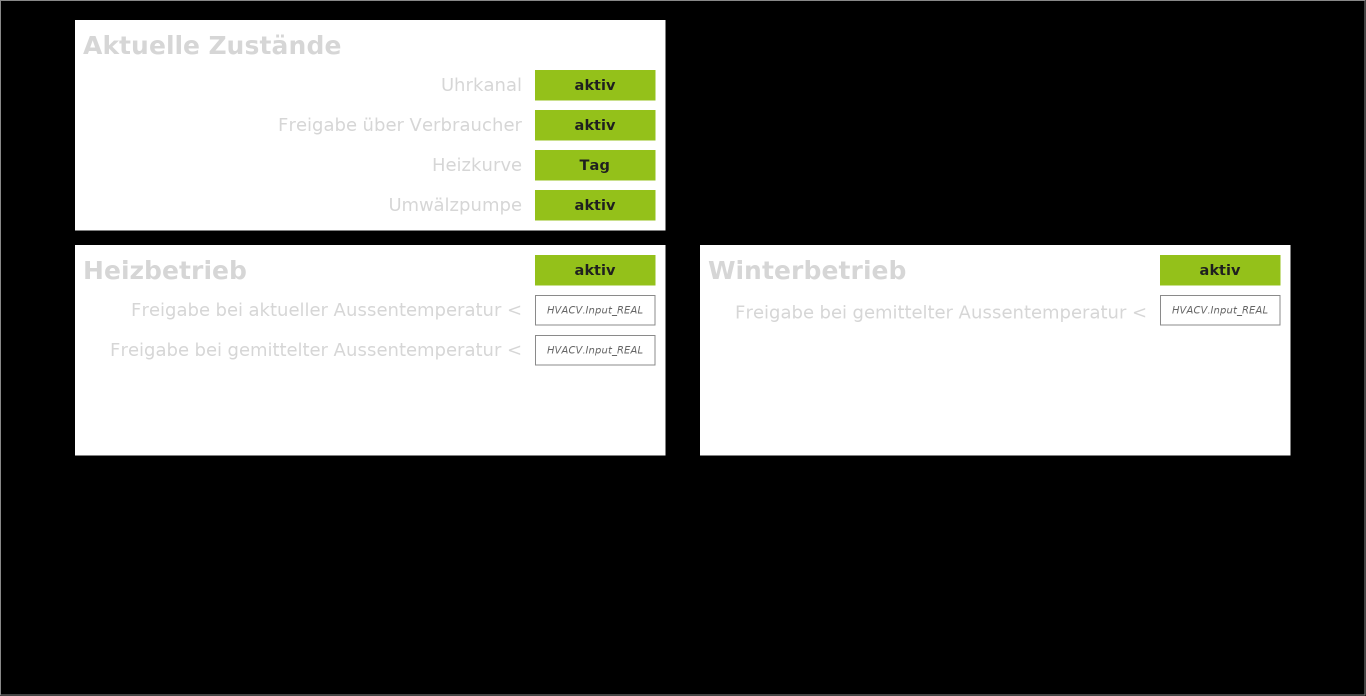
VISUALIZATION HeatingCircuit_VenA_Settings  // 1366x696
VAR_IN_OUT
	FB : HeatingCircuit_VenA;
END_VAR
    Rectangle (75,245 590x210)
    Rectangle (80,250 435x40), "Heizbetrieb"
    Rectangle (75,295 450x30), "Freigabe bei aktueller Aussentemperatur <"
    Rectangle (75,335 450x30), "Freigabe bei gemittelter Aussentemperatur <"
    RoundedRectangle (535,255 120x30), "inaktiv", invisible if: FB.HEAT
    RoundedRectangle (535,255 120x30), "aktiv", invisible if: NOT FB.HEAT
    Rectangle (75,20 590x210)
    Rectangle (80,25 570x40), "Aktuelle Zustände"
    Rectangle (75,70 450x30), "Uhrkanal"
    Rectangle (75,110 450x30), "Freigabe über Verbraucher"
    RoundedRectangle (535,70 120x30), "inaktiv", invisible if: FB.Clock_Channel
    RoundedRectangle (535,70 120x30), "aktiv", invisible if: NOT FB.Clock_Channel
    RoundedRectangle (535,110 120x30), "inaktiv", invisible if: FB.EXT_REQ
    RoundedRectangle (535,110 120x30), "aktiv", invisible if: NOT FB.EXT_REQ
    Rectangle (75,150 450x30), "Heizkurve"
    Rectangle (75,190 450x30), "Umwälzpumpe"
    RoundedRectangle (535,150 120x30), "Nacht", invisible if: FB.MODE
    RoundedRectangle (535,150 120x30), "Tag", invisible if: NOT FB.MODE
    RoundedRectangle (535,190 120x30), "inaktiv", invisible if: FB.pump.xAB
    RoundedRectangle (535,190 120x30), "aktiv", invisible if: NOT FB.pump.xAB
    Line (75,225)
    Line (965,345)
    Rectangle (700,245 590x210)
    Rectangle (705,250 435x40), "Winterbetrieb"
    Rectangle (700,295 450x35), "Freigabe bei gemittelter Aussentemperatur <"
    RoundedRectangle (1160,255 120x30), "inaktiv", invisible if: FB.WINTER
    RoundedRectangle (1160,255 120x30), "aktiv", invisible if: NOT FB.WINTER
    Frame (535,295 120x30)
        shows HVACV.Input_REAL(rValue := FB.Setpoint_Heat_Act.rSetPoint, bDecimals := 1, sUnit := '°C', rMinInputVisu := -20, rMaxInputVisu := 50, sDialogTitle := 'Release actual outsidetemp.')
    Frame (535,335 120x30)
        shows HVACV.Input_REAL(rValue := FB.Setpoint_Heat_Aver.rSetPoint, bDecimals := 1, sUnit := '°C', rMinInputVisu := -20, rMaxInputVisu := 50, sDialogTitle := 'Release average outsidetemp.')
    Frame (1160,295 120x30)
        shows HVACV.Input_REAL(rValue := FB.Setpoint_WINTER.rSetPoint, bDecimals := 1, sUnit := '°C', rMinInputVisu := -20, rMaxInputVisu := 50, sDialogTitle := 'Release winter operation')
END_VISUALIZATION

// Device/Application/Macros and frames/HeatingCircuit/Pump_Frames/Pump_Button
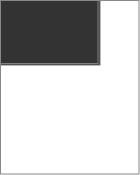
VISUALIZATION Pump_Button  // 140x175
VAR_IN_OUT
	FB_Pump : HVAC.Pump;
END_VAR

VAR 
	
END_VAR
    Rectangle (0,0 100x65), invisible if: TRUE
    Button (0,0 100x65)
        OnMouseClick:  Dialog=Pump_Parameter_Dialog, Parameters={FB_Pump: FB_Pump}, Selected={1: }, OpenModal=True, OpenCentered=True
END_VISUALIZATION

// Device/Application/Visu/1_Objects/HC_1/Heatcurve_HC_1
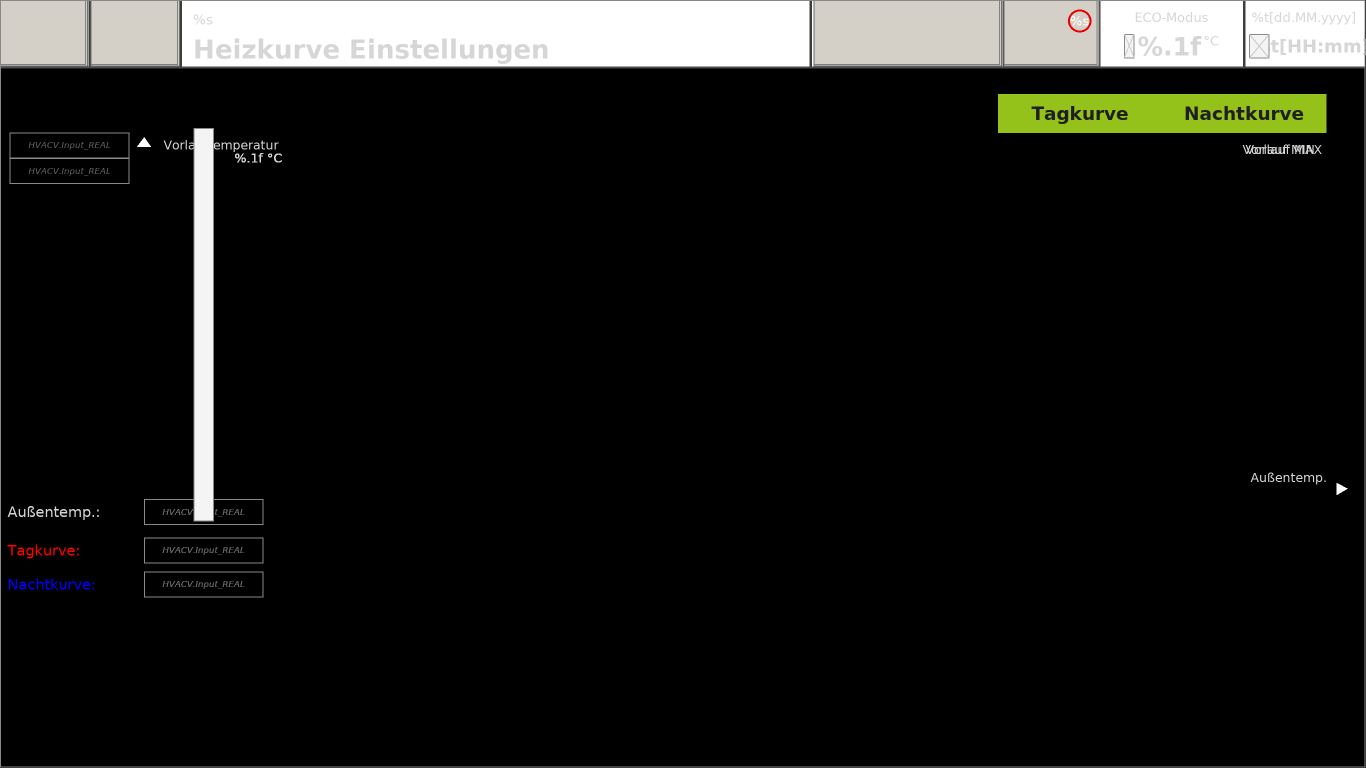
VISUALIZATION Heatcurve_HC_1  // 1366x768
    Frame (0,0 1366x70)
        shows Header_Frame()
    Rectangle (190,5 545x30), "%s", text variable: CONCAT( CONCAT(PRG.GebVar, ' | Start | Objekte | '), Prg.HC_1.Title)
    Rectangle (190,32 545x35), "Heizkurve Einstellungen"
    Frame (0,90 1357x595)
        shows HeatCurve4P_DN(FB_HeatCurve4P_DN := PRG.HC_1.HC)
END_VISUALIZATION

// Device/Application/Visu/1_Objects/HC_1/Trend_HC_1
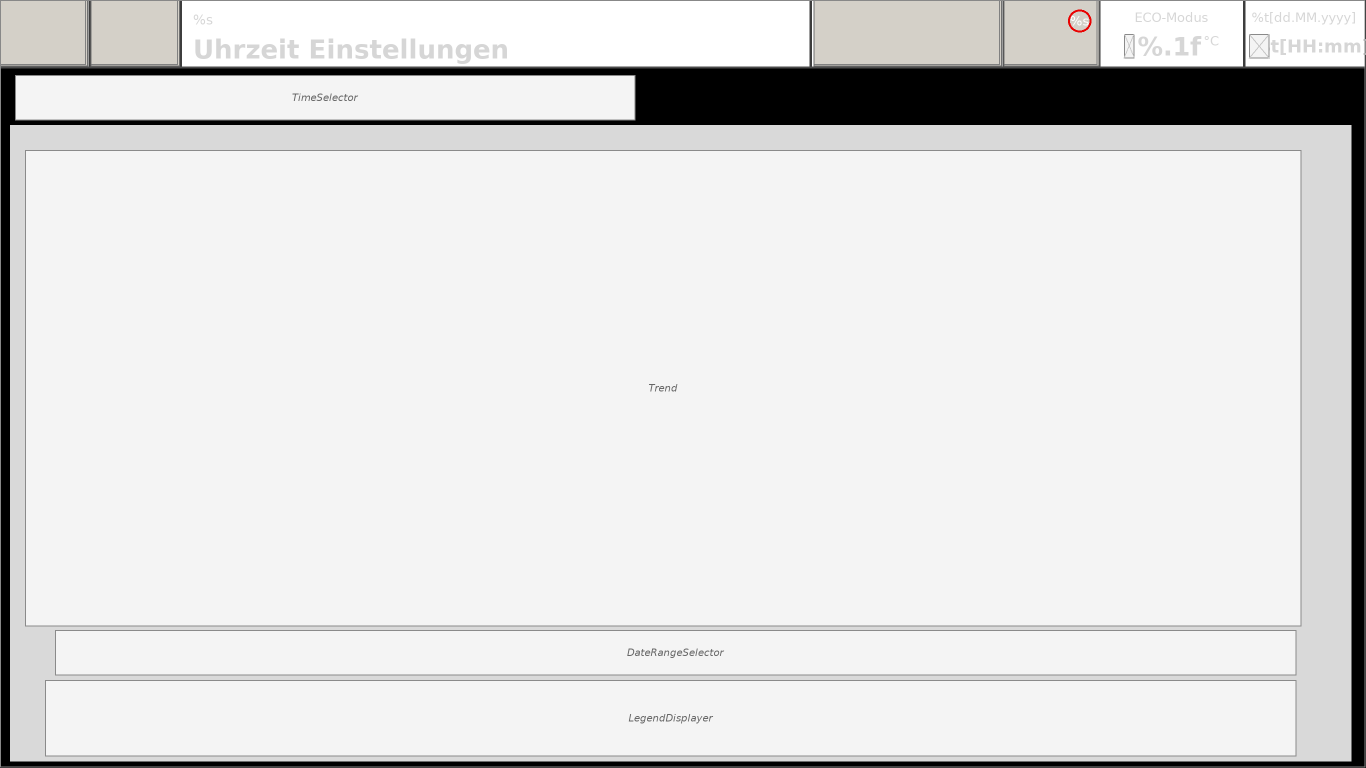
VISUALIZATION Trend_HC_1  // 1366x768
    Rectangle (10,125 1341x636)
    Frame (0,0 1366x70)
        shows Header_Frame()
    Rectangle (190,5 545x30), "%s", text variable: CONCAT( CONCAT(PRG.GebVar, ' | Start | Objekte | '), Prg.HC_1.Title)
    Rectangle (190,32 545x35), "Uhrzeit Einstellungen", text variable: PRG.HC_1.Title
    Trend (25,150 1276x476)
        p758368661: dd.MM.yyyy
        p2423372160: HH:mm
        p2833066001: HC_1_Trend
        p2059293862: Trend1DateRangeSelector
        p2541140726: Trend1TimeSelector
        p1690078355: Trend1Legend
    DateRangeSelector (55,630 1241x45)
        p758368661: dd.MM
        p2423372160: HH:mm
        p1661464551: GenElemInst_54
    TimeSelector (15,75 620x45)
        p3737533738: GenElemInst_54
        p677259794: Zoom:
    LegendDisplayer (45,680 1251x76)
        p3773266362: GenElemInst_54
END_VISUALIZATION

// Device/Application/Visu/3_Settings/Settings_MANInfo
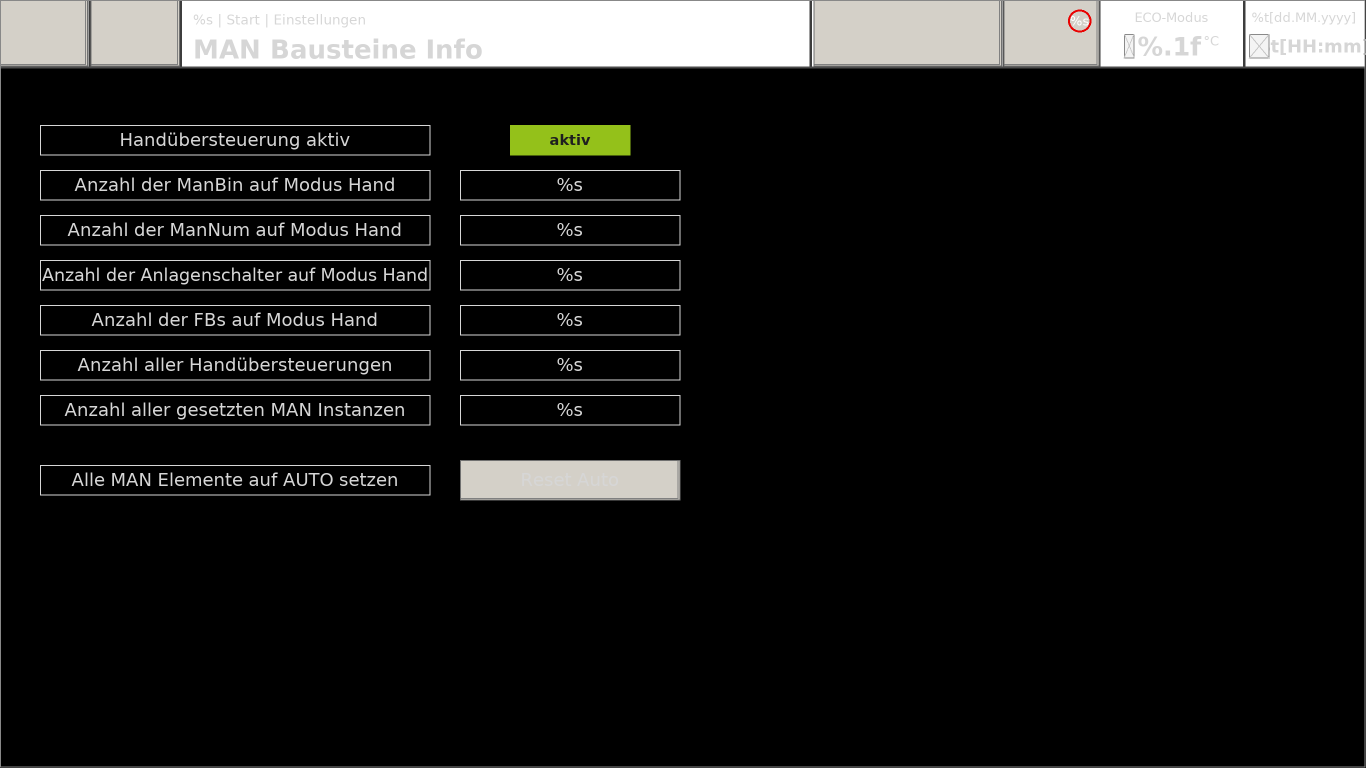
VISUALIZATION Settings_MANInfo  // 1366x768
    Rectangle (460,170 220x30), "%s", text variable: Main.ManInfo.iManBinCounter
    Rectangle (460,215 220x30), "%s", text variable: Main.ManInfo.iManNumCounter
    Rectangle (460,260 220x30), "%s", text variable: Main.ManInfo.iManOpCounter
    Rectangle (460,305 220x30), "%s", text variable: Main.ManInfo.iManFbCounter
    Rectangle (460,395 220x30), "%s", text variable: Main.ManInfo.iManCounter
    Rectangle (40,125 390x30), "Handübersteuerung aktiv"
    Rectangle (40,170 390x30), "Anzahl der ManBin auf Modus Hand"
    Rectangle (40,215 390x30), "Anzahl der ManNum auf Modus Hand"
    Rectangle (40,260 390x30), "Anzahl der Anlagenschalter auf Modus Hand"
    Rectangle (40,305 390x30), "Anzahl der FBs auf Modus Hand"
    Rectangle (40,395 390x30), "Anzahl aller gesetzten MAN Instanzen"
    Button (460,460 220x40), "Reset Auto"
        toggle Main.ManInfo.xResetAuto
    Frame (0,0 1366x70)
        shows Header_Frame()
    Rectangle (190,5 545x30), "%s | Start | Einstellungen", text variable: PRG.GebVar
    Rectangle (190,32 545x35), "MAN Bausteine Info"
    RoundedRectangle (510,125 120x30), "inaktiv", invisible if: Main.ManInfo.xManActive
    RoundedRectangle (510,125 120x30), "aktiv", invisible if: NOT Main.ManInfo.xManActive
    Rectangle (460,350 220x30), "%s", text variable: Main.ManInfo.iManCounter
    Rectangle (40,350 390x30), "Anzahl aller Handübersteuerungen"
    Rectangle (40,465 390x30), "Alle MAN Elemente auf AUTO setzen"
END_VISUALIZATION

// Device/Application/Visu/1_Objects/HC_1/Clock_HC_1
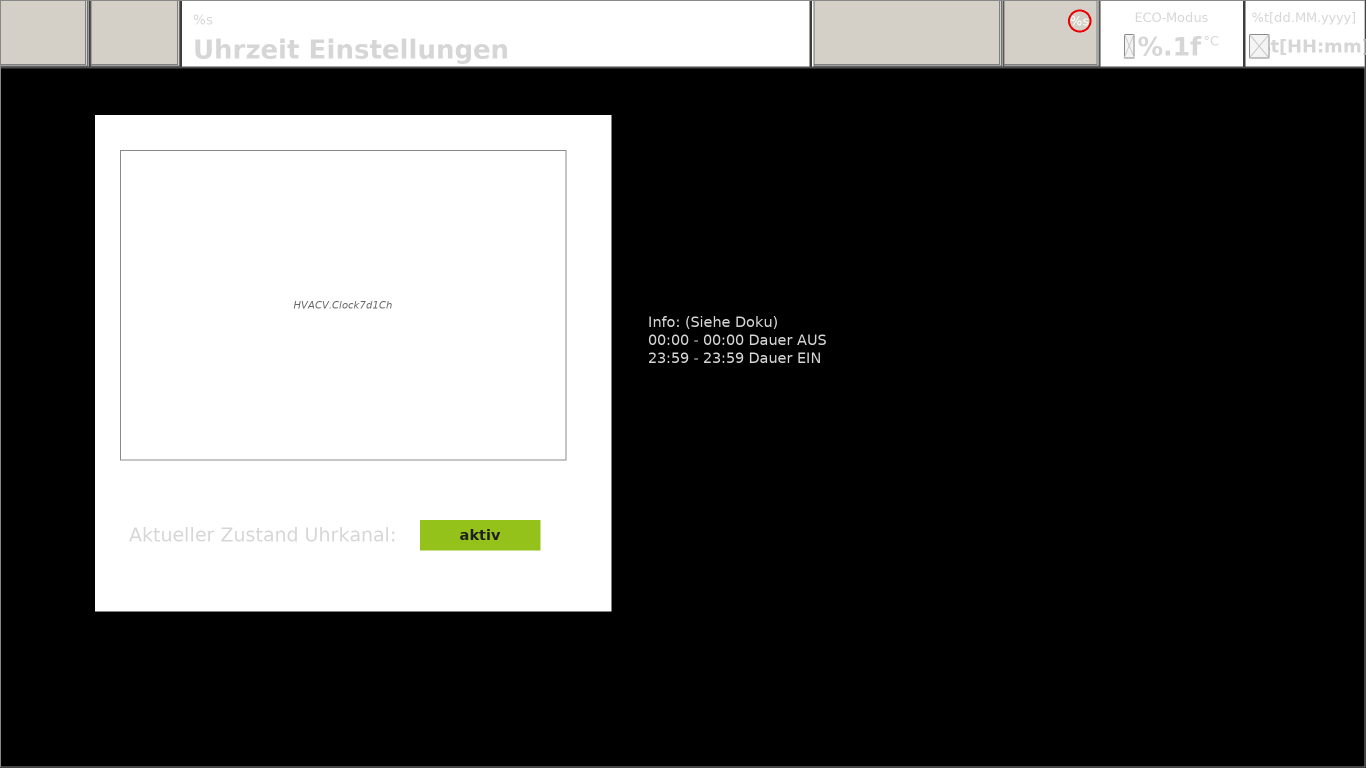
VISUALIZATION Clock_HC_1  // 1366x768
    Rectangle (95,115 516x496)
    Frame (0,0 1366x70)
        shows Header_Frame()
    Rectangle (190,5 545x30), "%s", text variable: CONCAT( CONCAT(PRG.GebVar, ' | Start | Objekte | '), Prg.HC_1.Title)
    Rectangle (190,32 545x35), "Uhrzeit Einstellungen", text variable: PRG.HC_1.Title
    RoundedRectangle (420,520 120x30), "inaktiv", invisible if: PRG.HC_1.Clock.xActive
    RoundedRectangle (420,520 120x30), "aktiv", invisible if: NOT PRG.HC_1.Clock.xActive
    Rectangle (115,520 296x30), "Aktueller Zustand Uhrkanal:"
    Frame (120,150 446x310)
        shows HVACV.Clock7d1Ch(FB_Clock7d1Ch := PRG.HC_1.Clock)
    Rectangle (645,295 447x90), "Info: (Siehe Doku) 00:00 - 00:00 Dauer AUS 23:59 - 23:59 Dauer EIN"
END_VISUALIZATION

// Device/Application/Visu/1_Objects/Room_1/Start_Room_1
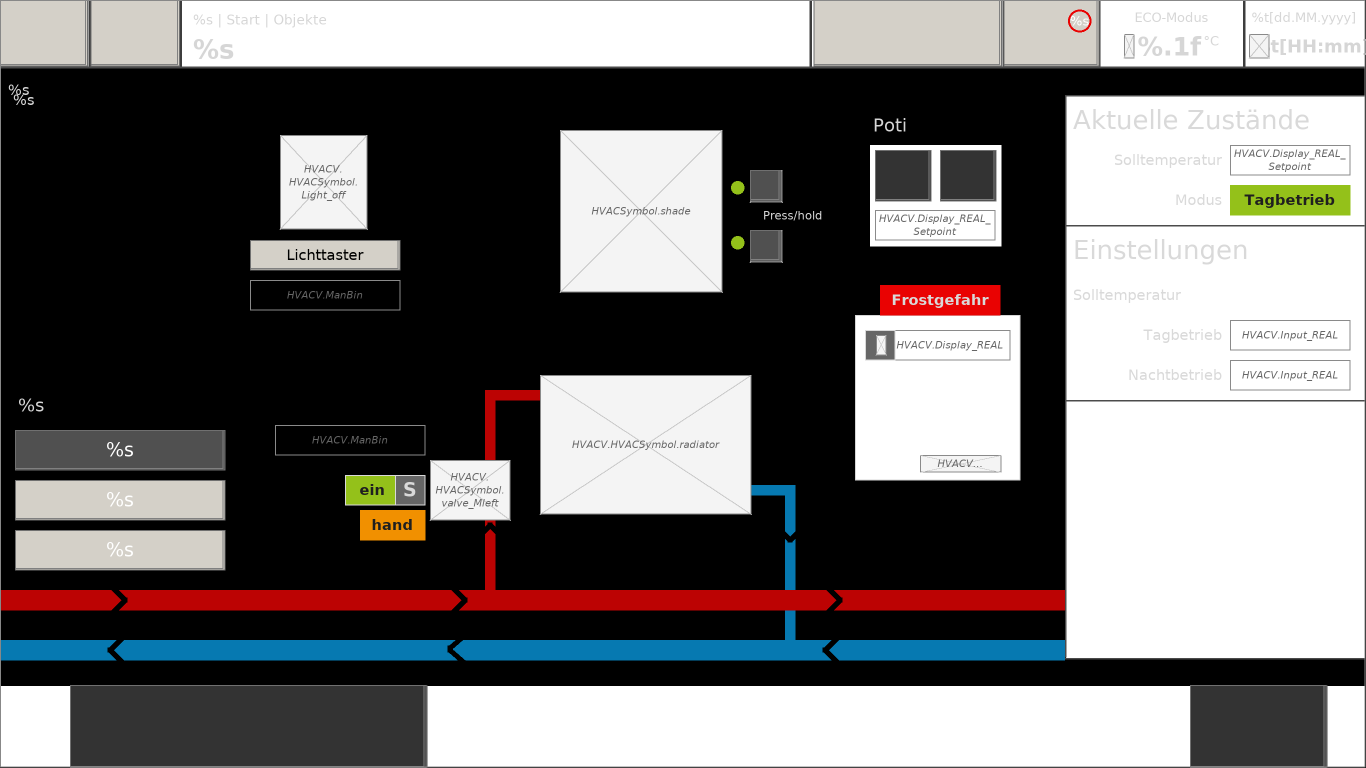
VISUALIZATION Start_Room_1  // 1366x768
    Frame (0,70 1366x613)
        shows Zone_F_Therm_Start(FB := PRG.Room_1)
    Frame (0,0 1366x70)
        shows Header_Frame()
    Rectangle (190,5 545x30), "%s | Start | Objekte", text variable: PRG.GebVar
    Rectangle (190,32 545x35), "%s", text variable: PRG.Room_1.Titel
    Rectangle (0,685 1366x83)
    Rectangle (425,685 2x83)
    Rectangle (70,685 2x83)
    Rectangle (130,685 166x83), "ZEITSCHALTUNG"
    Image (80,710 36x35), image: HVACV.HVACImage.clock
    RoundedRectangle (295,715 120x30), "inaktiv", invisible if: PRG.Room_1.Clock.xActive
    RoundedRectangle (295,715 120x30), "aktiv", invisible if: NOT PRG.Room_1.Clock.xActive
    Button (70,685 356x83)
        OnMouseClick:  Assign=Clock_Room_1, Type=Assignment
    Rectangle (1190,685 2x83)
    Rectangle (1325,685 2x83)
    Rectangle (1260,685 71x83), "HILFE"
    Image (1205,705 31x47), image: HVACV.HVACImage.help
    Button (1190,685 136x83)
        OnMouseClick:  Dialog=HVACV.Help_Start, OpenModal=True, OpenCentered=True
    Rectangle (10,85 536x30), "%s", text variable: PRG.Room_Line1.sSetPoint
        OnMouseClick: write the text variable via Default
END_VISUALIZATION

// Device/Application/Macros and frames/HeatingCircuit/Valve_Frames/ValveAnalog_Button
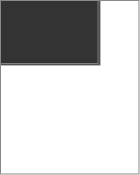
VISUALIZATION ValveAnalog_Button  // 140x175
VAR_IN_OUT
	FB_ValveAnalog : HVAC.ValveAnalog;
END_VAR

VAR 
	
END_VAR
    Rectangle (0,0 100x65), invisible if: TRUE
    Button (0,0 100x65)
        OnMouseClick:  Dialog=ValveAnalog_Parameter_Dialog, Parameters={FB_ValveAnalog: FB_ValveAnalog}, Selected={1: }, OpenModal=True, OpenCentered=True
END_VISUALIZATION

// Device/Application/Macros and frames/HeatingCircuit/HeatingCircuit_VenA
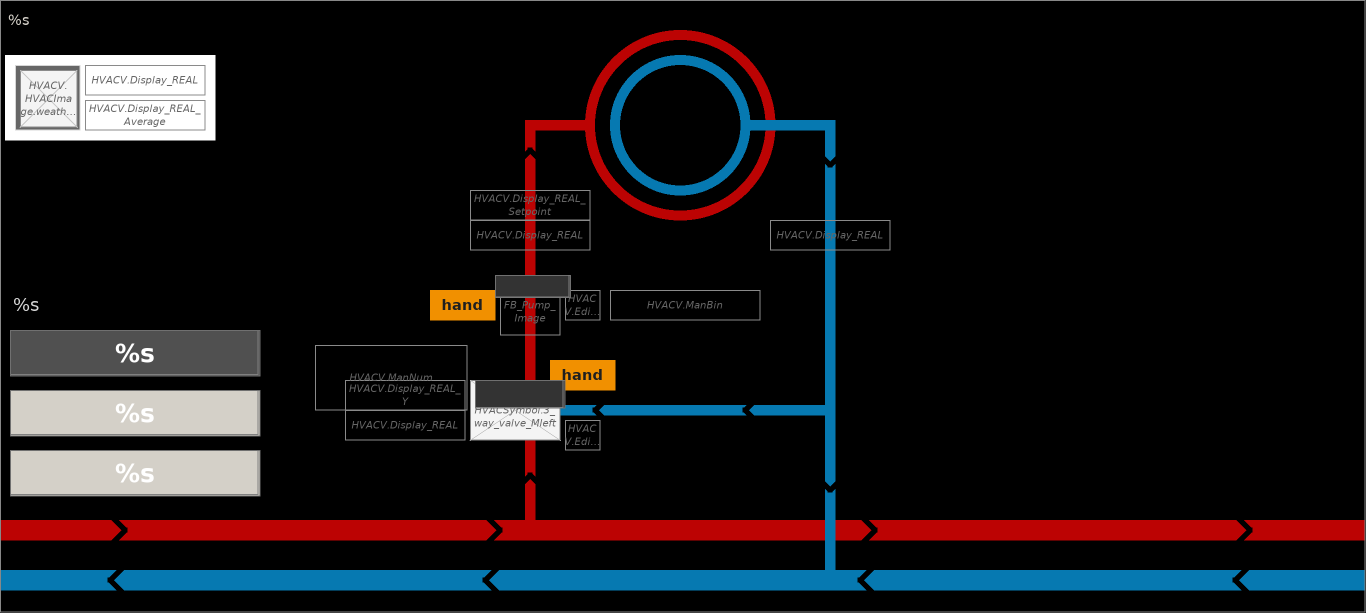
VISUALIZATION HeatingCircuit_VenA  // 1366x613
VAR_IN_OUT
	FB : HeatingCircuit_VenA;
END_VAR
    Rectangle (5,0 970x40), "%s", text variable: FB.Line1
    Rectangle (0,520 1365x20)
    Rectangle (0,570 1365x20)
    Polyline (875,565) (860,580) (875,595)
    Polyline (860,515) (875,530) (860,545)
    Polyline (125,565) (110,580) (125,595)
    Polyline (110,515) (125,530) (110,545)
    Polyline (485,515) (500,530) (485,545)
    Line (335,515)
    Polyline (1250,565) (1235,580) (1250,595)
    Polyline (1235,515) (1250,530) (1235,545)
    Rectangle (525,430 10x100)
    Rectangle (825,120 10x460)
    Rectangle (545,405 285x10)
    Rectangle (525,120 10x270)
    Polyline (515,490) (530,475) (545,490)
    Polyline (815,475) (830,490) (845,475)
    Polyline (815,150) (830,165) (845,150)
    Polyline (610,395) (595,410) (610,425)
    Polyline (760,395) (745,410) (760,425)
    Rectangle (525,120 65x10)
    Polyline (515,165) (530,150) (545,165)
    Image (470,380 90x60), image: HVACV.HVACSymbol.3_way_valve_Mleft
    Group (585,30 190x190)
        Ellipse (0,0 190x190)
        Ellipse (10,10 170x170)
        Ellipse (25,25 140x140)
        Ellipse (35,35 120x120)
    Rectangle (745,120 90x10)
    RoundedRectangle (430,290 65x30), "hand", invisible if: FB.Pump_AOO=0
    RoundedRectangle (550,360 65x30), "hand", invisible if: FB.Valve_AO = 0
    Frame (565,420 35x30)
        shows HVACV.Edit_symbol()
    Polyline (500,565) (485,580) (500,595)
    Frame (470,190 120x30)
        shows HVACV.Display_REAL_Setpoint(rSetpoint := FB.Setpoint_FT, bDecimals := 1, xAlarm := FALSE, sUnit := '°C')
    Frame (565,290 35x30)
        shows HVACV.Edit_symbol()
    Frame (500,275 60x60)
        shows HVACV.FB_Pump_Image(FB_Pump := FB.Pump)
    Rectangle (5,55 210x85)
    RoundedRectangle (15,65 65x65)
    Image (20,70 57x57), image: HVACV.HVACImage.weather
    Frame (85,100 120x30)
        shows HVACV.Display_REAL_Average(rValue := FB.OutTempAverage, bDecimals := 1, xAlarm := FALSE, sUnit := '°C')
    Frame (470,220 120x30)
        shows HVACV.Display_REAL(rValue := FB.TS_FT, bDecimals := 1, xAlarm := FB.TS_FT_ERR, sUnit := '°C')
    Frame (610,290 150x30)
        shows HVACV.ManBin(eManModeB := FB.Pump.eManModeB)
    Frame (85,65 120x30)
        shows HVACV.Display_REAL(rValue := FB.OutTemp, bDecimals := 1, xAlarm := FALSE, sUnit := '°C')
    Frame (770,220 120x30)
        shows HVACV.Display_REAL(rValue := FB.TS_RT, bDecimals := 1, xAlarm := FB.TS_RT_ERR, sUnit := '°C')
    Button (10,330 250x46), "%s", text variable: FB.OS.sTitleM0, colour toggle: FB.OS.eMode = 0
        OnMouseClick: execute { FB.OS.eMode := 0; }
    Button (10,390 250x46), "%s", text variable: FB.OS.sTitleM1, colour toggle: FB.OS.eMode =1
        OnMouseClick: execute { FB.OS.eMode := 1; }
    Button (10,450 250x46), "%s", text variable: FB.OS.sTitleM2, colour toggle: FB.OS.eMode =2
        OnMouseClick: execute { FB.OS.eMode := 2; }
    Frame (495,275 106x61)
        shows Pump_Button(FB_Pump := FB.Pump)
    Rectangle (10,290 250x30), "%s", text variable: FB.OS.sTitle
    Frame (475,380 126x76)
        shows ValveAnalog_Button(FB_ValveAnalog := FB.Valve)
    Frame (345,380 120x30)
        shows HVACV.Display_REAL_Y(rValue := FB.Valve_HA, bDecimals := 1, sUnit := '%')
    Frame (345,410 120x30)
        shows HVACV.Display_REAL(rValue := FB.Valve_rU, bDecimals := 1, xAlarm := FB.Valve.xAlarm, sUnit := '%')
    Frame (315,345 152x65)
        shows HVACV.ManNum(eManModeN := FB.Valve.eManModeN, rManValue := FB.Valve.rManValue, bDecimals := 1, sUnit := '%', rMinInputVisu := 0, rMaxInputVisu := 100, sDialogTitle := 'Manual valve position')
END_VISUALIZATION

// Device/Application/Visu/1_Objects/HC_1/Start_HC_1
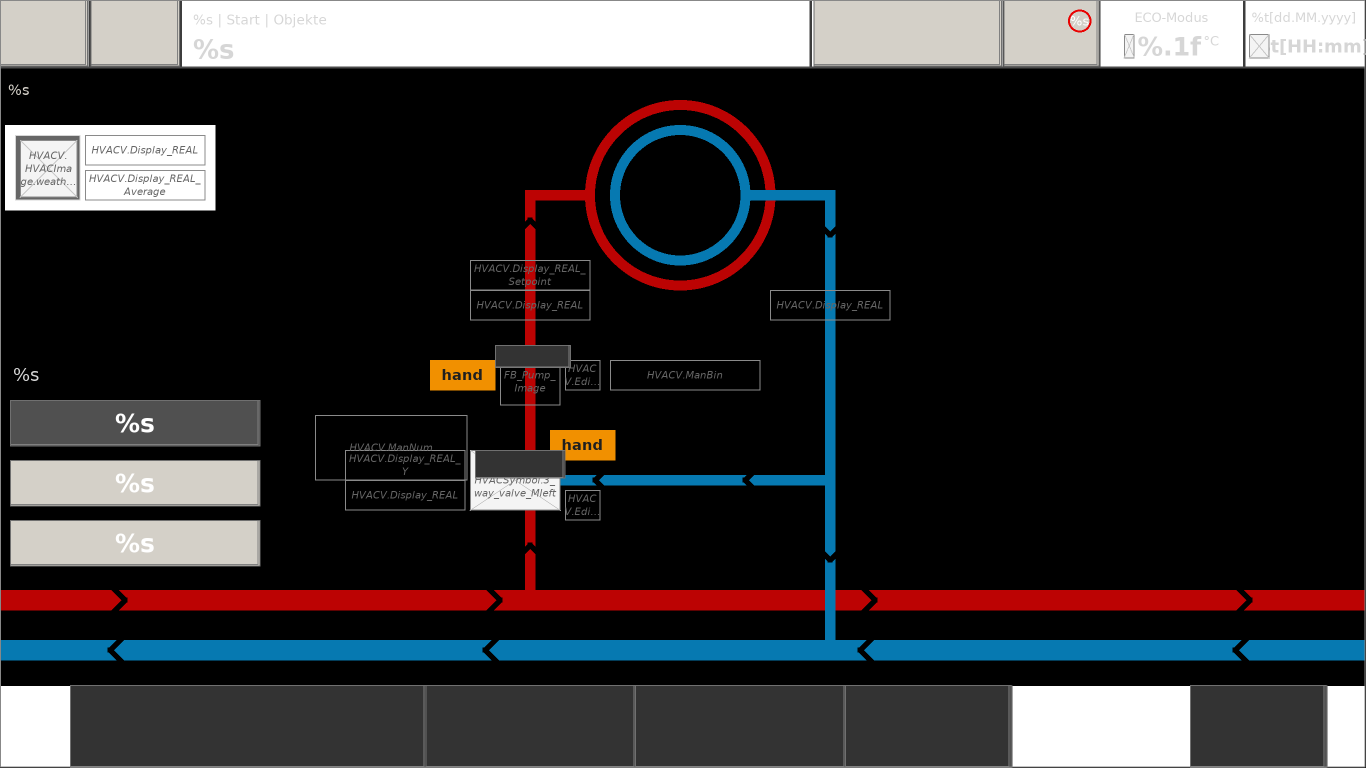
VISUALIZATION Start_HC_1  // 1366x768
    Frame (0,0 1366x70)
        shows Header_Frame()
    Rectangle (190,5 545x30), "%s | Start | Objekte", text variable: PRG.GebVar
    Rectangle (190,32 545x35), "%s", text variable: PRG.HC_1.Title
    Rectangle (0,685 1366x83)
    Rectangle (635,685 2x83)
    Rectangle (425,685 2x83)
    Rectangle (500,685 135x83), "EINSTELLUNG"
    Image (440,705 46x36), image: HVACV.HVACImage.settings
    Button (425,685 211x83)
        OnMouseClick:  Assign=Settings_HC_1, Type=Assignment
    Frame (0,70 1366x613)
        shows HeatingCircuit_VenA(FB := PRG.HC_1)
    Rectangle (70,685 2x83)
    Rectangle (130,685 166x83), "ZEITSCHALTUNG"
    Image (80,710 36x35), image: HVACV.HVACImage.clock
    Rectangle (705,685 136x83), "HEIZKURVE"
    Image (650,705 41x41), image: HVACV.HVACImage.heating_curve
    Button (635,685 211x83)
        OnMouseClick:  Assign=Heatcurve_HC_1, Type=Assignment
    RoundedRectangle (295,710 120x30), "inaktiv", invisible if: PRG.HC_1.Clock.xActive
    RoundedRectangle (295,710 120x30), "aktiv", invisible if: NOT PRG.HC_1.Clock.xActive
    Button (70,685 356x83)
        OnMouseClick:  Assign=Clock_HC_1, Type=Assignment
    Rectangle (1190,685 2x83)
    Rectangle (1325,685 2x83)
    Rectangle (1260,685 71x83), "HILFE"
    Image (1205,705 31x47), image: HVACV.HVACImage.help
    Button (1190,685 136x83)
        OnMouseClick:  Dialog=HVACV.Help_Start, OpenModal=True, OpenCentered=True
    Rectangle (845,685 2x83)
    Rectangle (1010,685 2x83)
    Rectangle (920,685 131x83), "TREND"
    Image (860,710 49x31), image: HVACV.HVACImage.trend
    Button (845,685 166x83)
        OnMouseClick:  Assign=Trend_HC_1, Type=Assignment
END_VISUALIZATION

// Device/Application/Macros and frames/HeatingCircuit/Pump_Frames/Pump_Parameter_Dialog
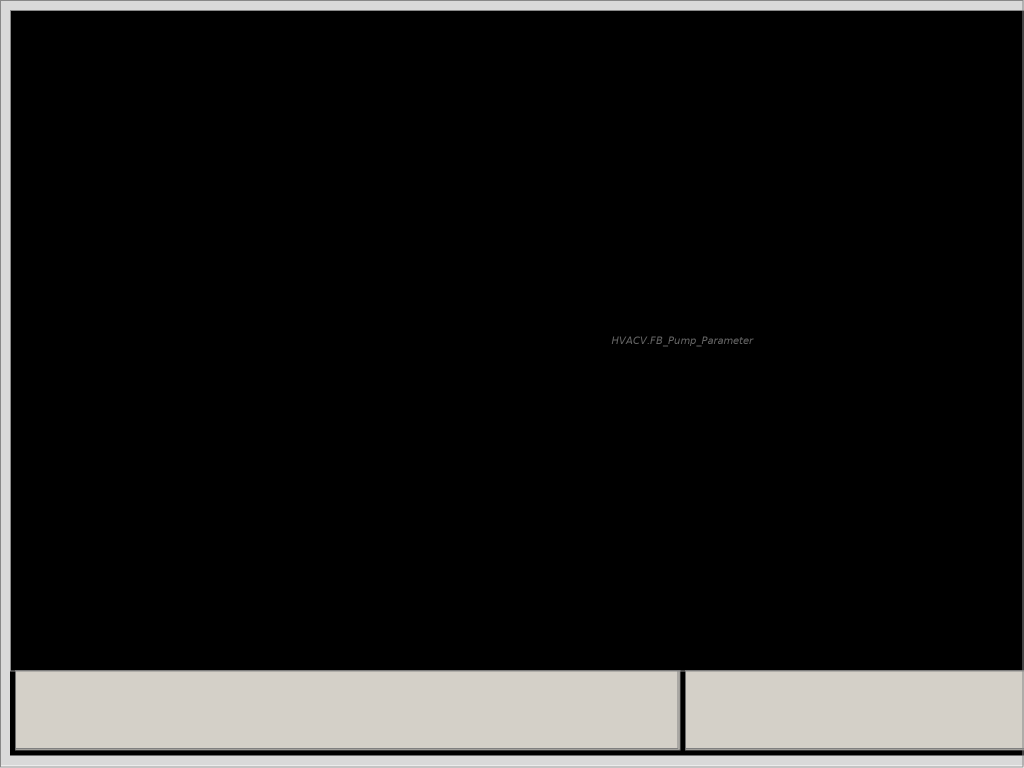
VISUALIZATION Pump_Parameter_Dialog  // 1024x768
VAR_IN_OUT
	FB_Pump : HVAC.Pump;
END_VAR
    Rectangle (0,0 1365x765)
    Rectangle (10,10 1345x745)
    Frame (685,670 665x80)
        shows HVACV.OK_Button(iPixel_Right := 365)
    Frame (15,670 665x80)
        shows HVACV.Exit_Button(iPixel_Right := 365)
    Button (685,670 665x80), tooltip "Schließen und Änderung übernehmen."
        OnMouseClick:  Dialog=Pump_Parameter_Dialog, Result=OK, NumpadKeypadSet=True
    Button (15,670 665x80)
        OnMouseClick:  Dialog=Pump_Parameter_Dialog, Result=Cancel, NumpadKeypadSet=True
    Frame (10,10 1345x661)
        shows HVACV.FB_Pump_Parameter(FB_Pump := FB_Pump)
    hotkey  Id=481037385728, Key=KeyDown=True, KeyName=ESCAPE, VisuElemId=264
    hotkey  Id=481038434304, Key=KeyName=ESCAPE, VisuElemId=264
    hotkey  Id=481039482880, Key=KeyDown=True, KeyName=RETURN_KEY, VisuElemId=266
    hotkey  Id=481040531456, Key=KeyName=RETURN_KEY, VisuElemId=266
END_VISUALIZATION

// Device/Application/Macros and frames/Clock/Holiday
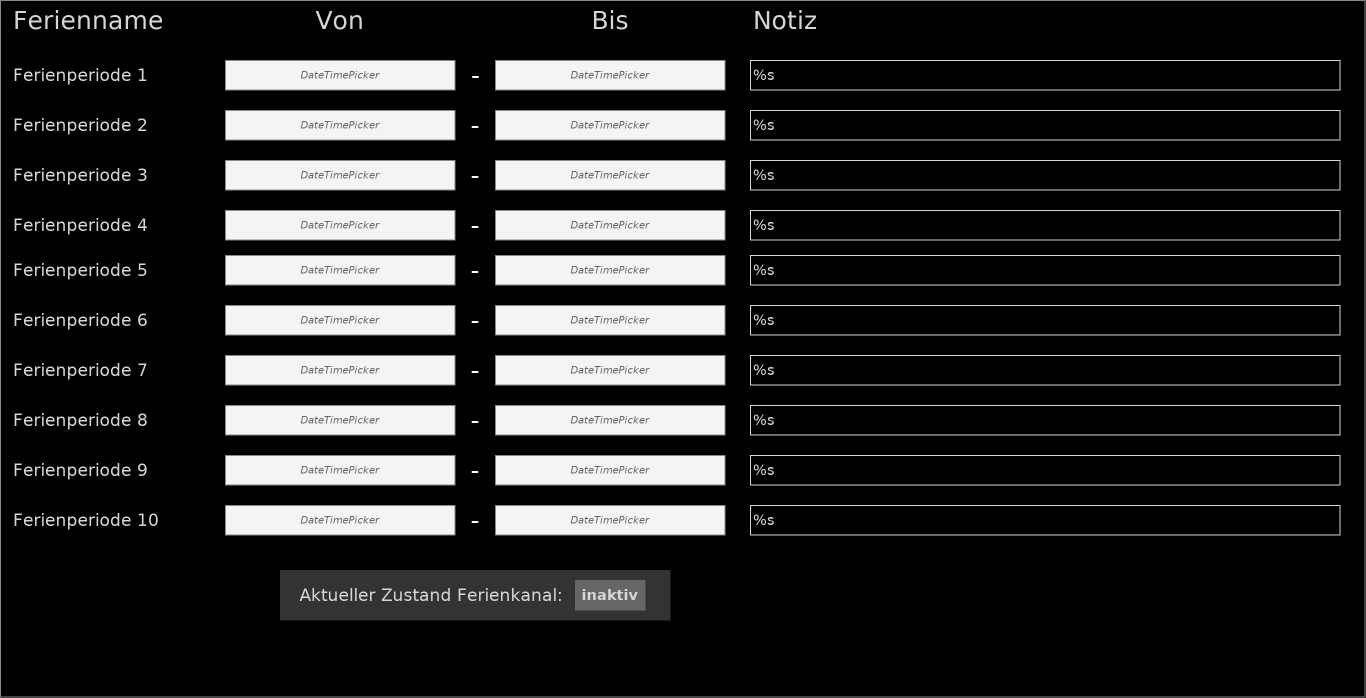
VISUALIZATION Holiday  // 1366x698
VAR_IN_OUT
	FB_Holiday : HVAC.Holiday;	
END_VAR
    Rectangle (225,60 230x30)
    Rectangle (10,60 180x30), "Ferienperiode 1"
    DateTimePicker (225,60 230x30)
        p2234502574: FB_Holiday.datCH1_DateFrom
        p1880513200: dd.MM.yyyy
    Rectangle (10,5 215x30), "Ferienname"
    Rectangle (225,5 230x30), "Von"
    Rectangle (495,5 230x30), "Bis"
    Rectangle (465,60 21x30), "-"
    Rectangle (10,110 180x30), "Ferienperiode 2"
    Rectangle (465,110 20x30), "-"
    Rectangle (10,160 180x30), "Ferienperiode 3"
    Rectangle (465,160 20x30), "-"
    Rectangle (10,210 180x30), "Ferienperiode 4"
    Rectangle (465,210 20x30), "-"
    Rectangle (10,255 180x30), "Ferienperiode 5"
    Rectangle (465,255 20x30), "-"
    Rectangle (10,305 180x30), "Ferienperiode 6"
    Rectangle (465,305 20x30), "-"
    Rectangle (10,355 180x30), "Ferienperiode 7"
    Rectangle (465,355 20x30), "-"
    Rectangle (10,405 180x30), "Ferienperiode 8"
    Rectangle (465,405 20x30), "-"
    Rectangle (10,455 180x30), "Ferienperiode 9"
    Rectangle (465,455 20x30), "-"
    Rectangle (10,505 180x30), "Ferienperiode 10"
    Rectangle (465,505 20x30), "-"
    Rectangle (750,60 590x30), "%s", text variable: FB_Holiday.sCH1_Notice
        OnMouseClick: write the text variable via Default
    Rectangle (750,110 590x30), "%s", text variable: FB_Holiday.sCH2_Notice
        OnMouseClick: write the text variable via Default
    Rectangle (750,160 590x30), "%s", text variable: FB_Holiday.sCH3_Notice
        OnMouseClick: write the text variable via Default
    Rectangle (750,210 590x30), "%s", text variable: FB_Holiday.sCH4_Notice
        OnMouseClick: write the text variable via Default
    Rectangle (750,255 590x30), "%s", text variable: FB_Holiday.sCH5_Notice
        OnMouseClick: write the text variable via Default
    Rectangle (750,305 590x30), "%s", text variable: FB_Holiday.sCH6_Notice
        OnMouseClick: write the text variable via Default
    Rectangle (750,355 590x30), "%s", text variable: FB_Holiday.sCH7_Notice
        OnMouseClick: write the text variable via Default
    Rectangle (750,405 590x30), "%s", text variable: FB_Holiday.sCH8_Notice
        OnMouseClick: write the text variable via Default
    Rectangle (750,455 590x30), "%s", text variable: FB_Holiday.sCH9_Notice
        OnMouseClick: write the text variable via Default
    Rectangle (750,505 590x30), "%s", text variable: FB_Holiday.sCH10_Notice
        OnMouseClick: write the text variable via Default
    Rectangle (750,5 510x30), "Notiz"
    Rectangle (280,570 390x50), "Aktueller Zustand Ferienkanal:"
    RoundedRectangle (585,580 50x30), "aktiv", invisible if: NOT(FB_Holiday.xActive)
    RoundedRectangle (575,580 70x30), "inaktiv", invisible if: FB_Holiday.xActive
    Rectangle (495,60 230x30)
    DateTimePicker (495,60 230x30)
        p2234502574: FB_Holiday.datCH1_DateTo
        p1880513200: dd.MM.yyyy
    Rectangle (225,110 230x30)
    DateTimePicker (225,110 230x30)
        p2234502574: FB_Holiday.datCH2_DateFrom
        p1880513200: dd.MM.yyyy
    Rectangle (495,110 230x30)
    DateTimePicker (495,110 230x30)
        p2234502574: FB_Holiday.datCH2_DateTo
        p1880513200: dd.MM.yyyy
    Rectangle (225,160 230x30)
    DateTimePicker (225,160 230x30)
        p2234502574: FB_Holiday.datCH3_DateFrom
        p1880513200: dd.MM.yyyy
    Rectangle (495,160 230x30)
    DateTimePicker (495,160 230x30)
        p2234502574: FB_Holiday.datCH3_DateTo
        p1880513200: dd.MM.yyyy
    Rectangle (225,210 230x30)
    DateTimePicker (225,210 230x30)
        p2234502574: FB_Holiday.datCH4_DateFrom
        p1880513200: dd.MM.yyyy
    Rectangle (495,210 230x30)
    DateTimePicker (495,210 230x30)
        p2234502574: FB_Holiday.datCH4_DateTo
        p1880513200: dd.MM.yyyy
    Rectangle (225,255 230x30)
    DateTimePicker (225,255 230x30)
        p2234502574: FB_Holiday.datCH5_DateFrom
        p1880513200: dd.MM.yyyy
    Rectangle (495,255 230x30)
    DateTimePicker (495,255 230x30)
        p2234502574: FB_Holiday.datCH5_DateTo
        p1880513200: dd.MM.yyyy
    Rectangle (225,305 230x30)
    DateTimePicker (225,305 230x30)
        p2234502574: FB_Holiday.datCH6_DateFrom
        p1880513200: dd.MM.yyyy
    Rectangle (495,305 230x30)
    DateTimePicker (495,305 230x30)
        p2234502574: FB_Holiday.datCH7_DateTo
        p1880513200: dd.MM.yyyy
    Rectangle (225,355 230x30)
    DateTimePicker (225,355 230x30)
        p2234502574: FB_Holiday.datCH7_DateFrom
        p1880513200: dd.MM.yyyy
    Rectangle (495,355 230x30)
    DateTimePicker (495,355 230x30)
        p2234502574: FB_Holiday.datCH7_DateTo
        p1880513200: dd.MM.yyyy
    Rectangle (225,405 230x30)
    DateTimePicker (225,405 230x30)
        p2234502574: FB_Holiday.datCH8_DateFrom
        p1880513200: dd.MM.yyyy
    Rectangle (495,405 230x30)
    DateTimePicker (495,405 230x30)
        p2234502574: FB_Holiday.datCH8_DateTo
        p1880513200: dd.MM.yyyy
    Rectangle (225,455 230x30)
    DateTimePicker (225,455 230x30)
        p2234502574: FB_Holiday.datCH9_DateFrom
        p1880513200: dd.MM.yyyy
    Rectangle (495,455 230x30)
    DateTimePicker (495,455 230x30)
        p2234502574: FB_Holiday.datCH9_DateTo
        p1880513200: dd.MM.yyyy
    Rectangle (225,505 230x30)
    DateTimePicker (225,505 230x30)
        p2234502574: FB_Holiday.datCH10_DateFrom
        p1880513200: dd.MM.yyyy
    Rectangle (495,505 230x30)
    DateTimePicker (495,505 230x30)
        p2234502574: FB_Holiday.datCH10_DateTo
        p1880513200: dd.MM.yyyy
END_VISUALIZATION

// Device/Application/Visu/2_Clock Settings/Clock_Settings_Start
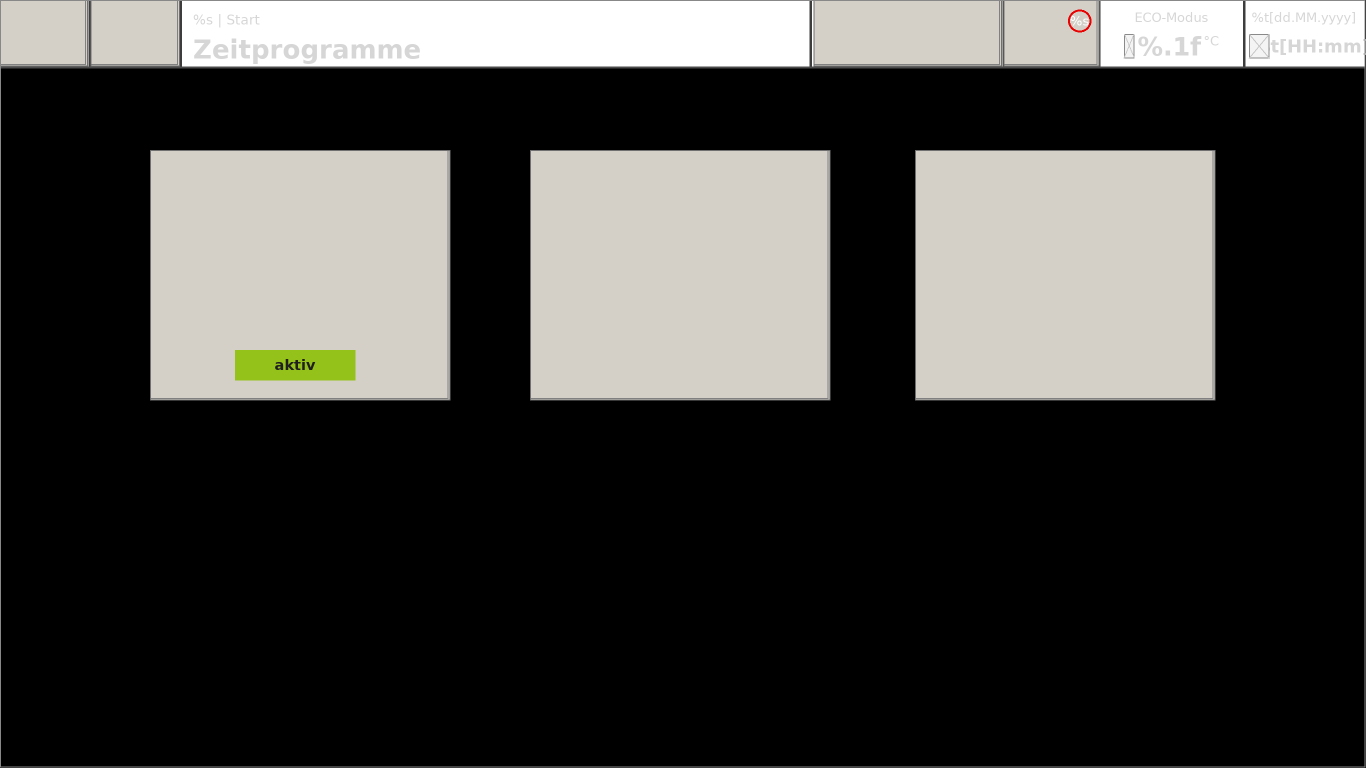
VISUALIZATION Clock_Settings_Start  // 1366x768
    Frame (0,0 1366x70)
        shows Header_Frame()
    Rectangle (190,5 545x30), "%s | Start", text variable: PRG.GebVar
    Rectangle (190,32 545x35), "Zeitprogramme"
    Rectangle (150,150 300x250)
    Rectangle (150,175 300x30), "FERIEN"
    Image (255,225 92x101), image: HVACV.HVACImage.calendar
    Button (150,150 300x250)
        OnMouseClick:  Assign=Clock_Holiday, Type=Assignment
    Rectangle (530,150 300x250)
    Rectangle (530,175 300x30), "FEIERTAGE"
    Image (625,225 110x96), image: HVACV.HVACImage.holiday
    RoundedRectangle (620,350 120x30), "inaktiv", invisible if: PRG.PublicHoliday_Demo.xActive
    RoundedRectangle (620,350 120x30), "aktiv", invisible if: NOT PRG.PublicHoliday_Demo.xActive
    Button (530,150 300x250)
        OnMouseClick:  Assign=Clock_Public_Holiday, Type=Assignment
    RoundedRectangle (235,350 120x30), "inaktiv", invisible if: PRG.Holiday_Demo.xActive
    RoundedRectangle (235,350 120x30), "aktiv", invisible if: NOT PRG.Holiday_Demo.xActive
    Rectangle (915,150 300x250)
    Rectangle (915,175 300x30), "SONDERZEITEN"
    Image (1015,225 93x103), image: HVACV.HVACImage.clock2
    RoundedRectangle (1005,350 120x30), "inaktiv", invisible if: PRG.SwitchTimeS_Demo.xActive
    RoundedRectangle (1005,350 120x30), "aktiv", invisible if: NOT PRG.SwitchTimeS_Demo.xActive
    Button (915,150 300x250)
        OnMouseClick:  Assign=Clock_SwitchTimeS, Type=Assignment
END_VISUALIZATION

// Device/Application/Macros and frames/Clock/PublicHoliday
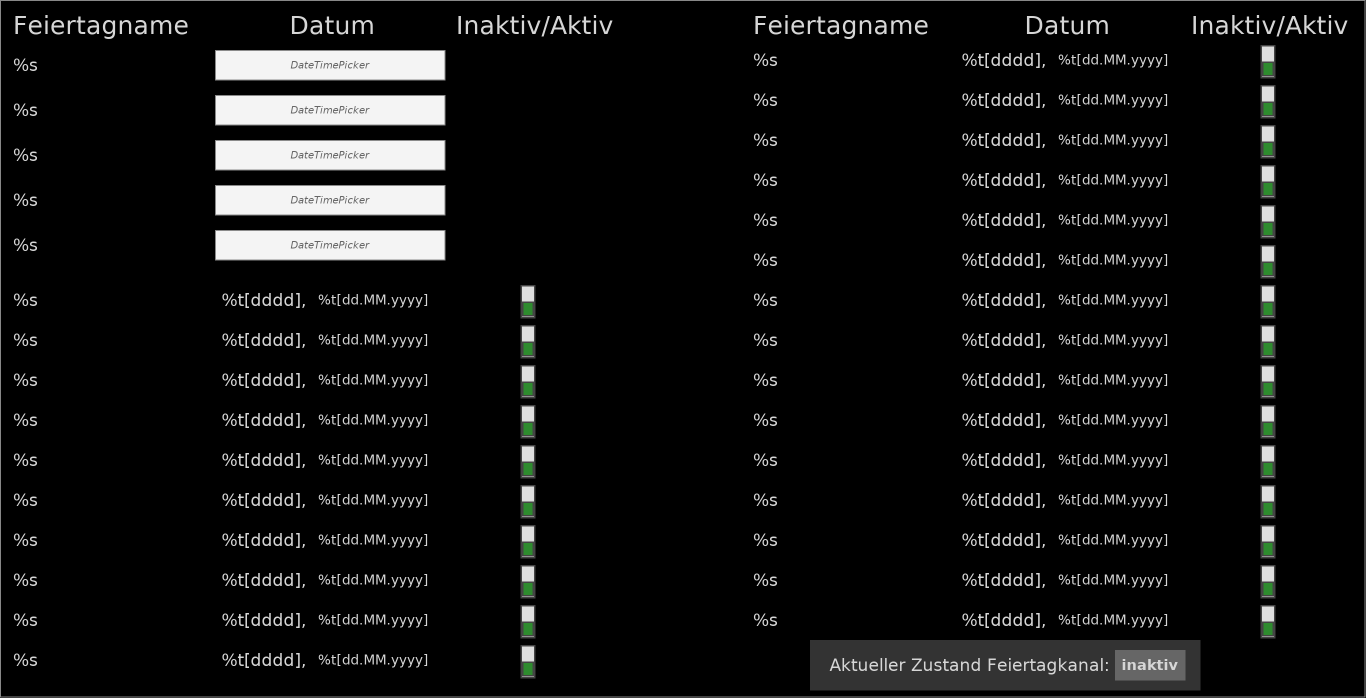
VISUALIZATION PublicHoliday  // 1366x698
VAR_IN_OUT
	FB_PublicHoliday : HVAC.PublicHoliday;	
END_VAR
    Rectangle (10,285 195x30), "%s", text variable: FB_PublicHoliday.astPublicHoliday[0].sName
    Rectangle (200,285 115x30), "%t[dddd],", text variable: FB_PublicHoliday.astPublicHoliday[0].datDate
    Rectangle (315,285 110x30), "%t[dd.MM.yyyy]", text variable: FB_PublicHoliday.astPublicHoliday[0].datDate
    Rectangle (230,10 205x30), "Datum"
    Rectangle (450,10 170x30), "Inaktiv/Aktiv"
    Rectangle (10,50 215x30), "%s", text variable: FB_PublicHoliday.astPublicHoliday[25].sName
        OnMouseClick: write the text variable via Default
    DipSwitch (495,285 66x33), variable: FB_PublicHoliday.astPublicHoliday[0].xEnable, behaviour: TOGGLE, style: Switch-DipSwitch-Green
    Rectangle (10,325 195x30), "%s", text variable: FB_PublicHoliday.astPublicHoliday[1].sName
    Rectangle (200,325 115x30), "%t[dddd],", text variable: FB_PublicHoliday.astPublicHoliday[1].datDate
    Rectangle (315,325 110x30), "%t[dd.MM.yyyy]", text variable: FB_PublicHoliday.astPublicHoliday[1].datDate
    DipSwitch (495,325 66x33), variable: FB_PublicHoliday.astPublicHoliday[1].xEnable, behaviour: TOGGLE, style: Switch-DipSwitch-Green
    Rectangle (10,365 195x30), "%s", text variable: FB_PublicHoliday.astPublicHoliday[2].sName
    Rectangle (200,365 115x30), "%t[dddd],", text variable: FB_PublicHoliday.astPublicHoliday[2].datDate
    Rectangle (315,365 110x30), "%t[dd.MM.yyyy]", text variable: FB_PublicHoliday.astPublicHoliday[2].datDate
    DipSwitch (495,365 66x33), variable: FB_PublicHoliday.astPublicHoliday[2].xEnable, behaviour: TOGGLE, style: Switch-DipSwitch-Green
    Rectangle (10,405 195x30), "%s", text variable: FB_PublicHoliday.astPublicHoliday[3].sName
    Rectangle (200,405 115x30), "%t[dddd],", text variable: FB_PublicHoliday.astPublicHoliday[3].datDate
    Rectangle (315,405 110x30), "%t[dd.MM.yyyy]", text variable: FB_PublicHoliday.astPublicHoliday[3].datDate
    DipSwitch (495,405 66x33), variable: FB_PublicHoliday.astPublicHoliday[3].xEnable, behaviour: TOGGLE, style: Switch-DipSwitch-Green
    Rectangle (10,445 195x30), "%s", text variable: FB_PublicHoliday.astPublicHoliday[4].sName
    Rectangle (200,445 115x30), "%t[dddd],", text variable: FB_PublicHoliday.astPublicHoliday[4].datDate
    Rectangle (315,445 110x30), "%t[dd.MM.yyyy]", text variable: FB_PublicHoliday.astPublicHoliday[4].datDate
    DipSwitch (495,445 66x33), variable: FB_PublicHoliday.astPublicHoliday[4].xEnable, behaviour: TOGGLE, style: Switch-DipSwitch-Green
    Rectangle (10,485 195x30), "%s", text variable: FB_PublicHoliday.astPublicHoliday[5].sName
    Rectangle (200,485 115x30), "%t[dddd],", text variable: FB_PublicHoliday.astPublicHoliday[5].datDate
    Rectangle (315,485 110x30), "%t[dd.MM.yyyy]", text variable: FB_PublicHoliday.astPublicHoliday[5].datDate
    DipSwitch (495,485 66x33), variable: FB_PublicHoliday.astPublicHoliday[5].xEnable, behaviour: TOGGLE, style: Switch-DipSwitch-Green
    Rectangle (10,525 195x30), "%s", text variable: FB_PublicHoliday.astPublicHoliday[6].sName
    Rectangle (200,525 115x30), "%t[dddd],", text variable: FB_PublicHoliday.astPublicHoliday[6].datDate
    Rectangle (315,525 110x30), "%t[dd.MM.yyyy]", text variable: FB_PublicHoliday.astPublicHoliday[6].datDate
    DipSwitch (495,525 66x33), variable: FB_PublicHoliday.astPublicHoliday[6].xEnable, behaviour: TOGGLE, style: Switch-DipSwitch-Green
    Rectangle (10,565 195x30), "%s", text variable: FB_PublicHoliday.astPublicHoliday[7].sName
    Rectangle (200,565 115x30), "%t[dddd],", text variable: FB_PublicHoliday.astPublicHoliday[7].datDate
    Rectangle (315,565 110x30), "%t[dd.MM.yyyy]", text variable: FB_PublicHoliday.astPublicHoliday[7].datDate
    DipSwitch (495,565 66x33), variable: FB_PublicHoliday.astPublicHoliday[7].xEnable, behaviour: TOGGLE, style: Switch-DipSwitch-Green
    Rectangle (10,605 195x30), "%s", text variable: FB_PublicHoliday.astPublicHoliday[8].sName
    Rectangle (200,605 115x30), "%t[dddd],", text variable: FB_PublicHoliday.astPublicHoliday[8].datDate
    Rectangle (315,605 110x30), "%t[dd.MM.yyyy]", text variable: FB_PublicHoliday.astPublicHoliday[8].datDate
    DipSwitch (495,605 66x33), variable: FB_PublicHoliday.astPublicHoliday[8].xEnable, behaviour: TOGGLE, style: Switch-DipSwitch-Green
    Rectangle (10,645 195x30), "%s", text variable: FB_PublicHoliday.astPublicHoliday[9].sName
    Rectangle (200,645 115x30), "%t[dddd],", text variable: FB_PublicHoliday.astPublicHoliday[9].datDate
    Rectangle (315,645 110x30), "%t[dd.MM.yyyy]", text variable: FB_PublicHoliday.astPublicHoliday[9].datDate
    DipSwitch (495,645 66x33), variable: FB_PublicHoliday.astPublicHoliday[9].xEnable, behaviour: TOGGLE, style: Switch-DipSwitch-Green
    Rectangle (750,45 195x30), "%s", text variable: FB_PublicHoliday.astPublicHoliday[10].sName
    Rectangle (940,45 115x30), "%t[dddd],", text variable: FB_PublicHoliday.astPublicHoliday[10].datDate
    Rectangle (1055,45 110x30), "%t[dd.MM.yyyy]", text variable: FB_PublicHoliday.astPublicHoliday[10].datDate
    DipSwitch (1235,45 66x33), variable: FB_PublicHoliday.astPublicHoliday[10].xEnable, behaviour: TOGGLE, style: Switch-DipSwitch-Green
    Rectangle (750,85 195x30), "%s", text variable: FB_PublicHoliday.astPublicHoliday[11].sName
    Rectangle (940,85 115x30), "%t[dddd],", text variable: FB_PublicHoliday.astPublicHoliday[11].datDate
    Rectangle (1055,85 110x30), "%t[dd.MM.yyyy]", text variable: FB_PublicHoliday.astPublicHoliday[11].datDate
    DipSwitch (1235,85 66x33), variable: FB_PublicHoliday.astPublicHoliday[11].xEnable, behaviour: TOGGLE, style: Switch-DipSwitch-Green
    Rectangle (750,125 195x30), "%s", text variable: FB_PublicHoliday.astPublicHoliday[12].sName
    Rectangle (940,125 115x30), "%t[dddd],", text variable: FB_PublicHoliday.astPublicHoliday[12].datDate
    Rectangle (1055,125 110x30), "%t[dd.MM.yyyy]", text variable: FB_PublicHoliday.astPublicHoliday[12].datDate
    DipSwitch (1235,125 66x33), variable: FB_PublicHoliday.astPublicHoliday[12].xEnable, behaviour: TOGGLE, style: Switch-DipSwitch-Green
    Rectangle (750,165 195x30), "%s", text variable: FB_PublicHoliday.astPublicHoliday[13].sName
    Rectangle (940,165 115x30), "%t[dddd],", text variable: FB_PublicHoliday.astPublicHoliday[13].datDate
    Rectangle (1055,165 110x30), "%t[dd.MM.yyyy]", text variable: FB_PublicHoliday.astPublicHoliday[13].datDate
    DipSwitch (1235,165 66x33), variable: FB_PublicHoliday.astPublicHoliday[13].xEnable, behaviour: TOGGLE, style: Switch-DipSwitch-Green
    Rectangle (750,205 195x30), "%s", text variable: FB_PublicHoliday.astPublicHoliday[14].sName
    Rectangle (940,205 115x30), "%t[dddd],", text variable: FB_PublicHoliday.astPublicHoliday[14].datDate
    Rectangle (1055,205 110x30), "%t[dd.MM.yyyy]", text variable: FB_PublicHoliday.astPublicHoliday[14].datDate
    DipSwitch (1235,205 66x33), variable: FB_PublicHoliday.astPublicHoliday[14].xEnable, behaviour: TOGGLE, style: Switch-DipSwitch-Green
    Rectangle (750,245 195x30), "%s", text variable: FB_PublicHoliday.astPublicHoliday[15].sName
    Rectangle (940,245 115x30), "%t[dddd],", text variable: FB_PublicHoliday.astPublicHoliday[15].datDate
    Rectangle (1055,245 110x30), "%t[dd.MM.yyyy]", text variable: FB_PublicHoliday.astPublicHoliday[15].datDate
    DipSwitch (1235,245 66x33), variable: FB_PublicHoliday.astPublicHoliday[15].xEnable, behaviour: TOGGLE, style: Switch-DipSwitch-Green
    Rectangle (750,285 195x30), "%s", text variable: FB_PublicHoliday.astPublicHoliday[16].sName
    Rectangle (940,285 115x30), "%t[dddd],", text variable: FB_PublicHoliday.astPublicHoliday[16].datDate
    Rectangle (1055,285 110x30), "%t[dd.MM.yyyy]", text variable: FB_PublicHoliday.astPublicHoliday[16].datDate
    DipSwitch (1235,285 66x33), variable: FB_PublicHoliday.astPublicHoliday[16].xEnable, behaviour: TOGGLE, style: Switch-DipSwitch-Green
    Rectangle (750,10 185x30), "Feiertagname"
    Rectangle (965,10 205x30), "Datum"
    Rectangle (1185,10 170x30), "Inaktiv/Aktiv"
    Rectangle (750,325 195x30), "%s", text variable: FB_PublicHoliday.astPublicHoliday[17].sName
    Rectangle (940,325 115x30), "%t[dddd],", text variable: FB_PublicHoliday.astPublicHoliday[17].datDate
    Rectangle (1055,325 110x30), "%t[dd.MM.yyyy]", text variable: FB_PublicHoliday.astPublicHoliday[17].datDate
    DipSwitch (1235,325 66x33), variable: FB_PublicHoliday.astPublicHoliday[17].xEnable, behaviour: TOGGLE, style: Switch-DipSwitch-Green
    Rectangle (750,365 195x30), "%s", text variable: FB_PublicHoliday.astPublicHoliday[18].sName
    Rectangle (940,365 115x30), "%t[dddd],", text variable: FB_PublicHoliday.astPublicHoliday[18].datDate
    Rectangle (1055,365 110x30), "%t[dd.MM.yyyy]", text variable: FB_PublicHoliday.astPublicHoliday[18].datDate
    DipSwitch (1235,365 66x33), variable: FB_PublicHoliday.astPublicHoliday[18].xEnable, behaviour: TOGGLE, style: Switch-DipSwitch-Green
    Rectangle (750,405 195x30), "%s", text variable: FB_PublicHoliday.astPublicHoliday[19].sName
    Rectangle (940,405 115x30), "%t[dddd],", text variable: FB_PublicHoliday.astPublicHoliday[19].datDate
    Rectangle (1055,405 110x30), "%t[dd.MM.yyyy]", text variable: FB_PublicHoliday.astPublicHoliday[19].datDate
    DipSwitch (1235,405 66x33), variable: FB_PublicHoliday.astPublicHoliday[19].xEnable, behaviour: TOGGLE, style: Switch-DipSwitch-Green
    Rectangle (750,445 195x30), "%s", text variable: FB_PublicHoliday.astPublicHoliday[20].sName
    Rectangle (940,445 115x30), "%t[dddd],", text variable: FB_PublicHoliday.astPublicHoliday[20].datDate
    Rectangle (1055,445 110x30), "%t[dd.MM.yyyy]", text variable: FB_PublicHoliday.astPublicHoliday[20].datDate
    DipSwitch (1235,445 66x33), variable: FB_PublicHoliday.astPublicHoliday[20].xEnable, behaviour: TOGGLE, style: Switch-DipSwitch-Green
    Rectangle (750,485 195x30), "%s", text variable: FB_PublicHoliday.astPublicHoliday[21].sName
    Rectangle (940,485 115x30), "%t[dddd],", text variable: FB_PublicHoliday.astPublicHoliday[21].datDate
    Rectangle (1055,485 110x30), "%t[dd.MM.yyyy]", text variable: FB_PublicHoliday.astPublicHoliday[21].datDate
    DipSwitch (1235,485 66x33), variable: FB_PublicHoliday.astPublicHoliday[21].xEnable, behaviour: TOGGLE, style: Switch-DipSwitch-Green
    Rectangle (750,525 195x30), "%s", text variable: FB_PublicHoliday.astPublicHoliday[22].sName
    Rectangle (940,525 115x30), "%t[dddd],", text variable: FB_PublicHoliday.astPublicHoliday[22].datDate
    Rectangle (1055,525 110x30), "%t[dd.MM.yyyy]", text variable: FB_PublicHoliday.astPublicHoliday[22].datDate
    DipSwitch (1235,525 66x33), variable: FB_PublicHoliday.astPublicHoliday[22].xEnable, behaviour: TOGGLE, style: Switch-DipSwitch-Green
    Rectangle (750,565 195x30), "%s", text variable: FB_PublicHoliday.astPublicHoliday[23].sName
    Rectangle (940,565 115x30), "%t[dddd],", text variable: FB_PublicHoliday.astPublicHoliday[23].datDate
    Rectangle (1055,565 110x30), "%t[dd.MM.yyyy]", text variable: FB_PublicHoliday.astPublicHoliday[23].datDate
    DipSwitch (1235,565 66x33), variable: FB_PublicHoliday.astPublicHoliday[23].xEnable, behaviour: TOGGLE, style: Switch-DipSwitch-Green
    Rectangle (750,605 195x30), "%s", text variable: FB_PublicHoliday.astPublicHoliday[24].sName
    Rectangle (940,605 115x30), "%t[dddd],", text variable: FB_PublicHoliday.astPublicHoliday[24].datDate
    Rectangle (1055,605 110x30), "%t[dd.MM.yyyy]", text variable: FB_PublicHoliday.astPublicHoliday[24].datDate
    DipSwitch (1235,605 66x33), variable: FB_PublicHoliday.astPublicHoliday[24].xEnable, behaviour: TOGGLE, style: Switch-DipSwitch-Green
    Rectangle (10,10 240x30), "Feiertagname"
    Rectangle (10,95 215x30), "%s", text variable: FB_PublicHoliday.astPublicHoliday[26].sName
        OnMouseClick: write the text variable via Default
    Rectangle (10,140 215x30), "%s", text variable: FB_PublicHoliday.astPublicHoliday[27].sName
        OnMouseClick: write the text variable via Default
    Rectangle (10,185 215x30), "%s", text variable: FB_PublicHoliday.astPublicHoliday[28].sName
        OnMouseClick: write the text variable via Default
    Rectangle (10,230 215x30), "%s", text variable: FB_PublicHoliday.astPublicHoliday[29].sName
        OnMouseClick: write the text variable via Default
    Rectangle (810,640 390x50), "Aktueller Zustand Feiertagkanal:"
    RoundedRectangle (1125,650 50x30), "aktiv", invisible if: NOT(FB_PublicHoliday.xActive)
    RoundedRectangle (1115,650 70x30), "inaktiv", invisible if: FB_PublicHoliday.xActive
    Rectangle (215,50 230x30)
    DateTimePicker (215,50 230x30)
        p2234502574: FB_PublicHoliday.astPublicHoliday[25].datDate
        p1880513200: dd.MM.yyyy
    Rectangle (215,95 230x30)
    DateTimePicker (215,95 230x30)
        p2234502574: FB_PublicHoliday.astPublicHoliday[26].datDate
        p1880513200: dd.MM.yyyy
    Rectangle (215,140 230x30)
    DateTimePicker (215,140 230x30)
        p2234502574: FB_PublicHoliday.astPublicHoliday[27].datDate
        p1880513200: dd.MM.yyyy
    Rectangle (215,185 230x30)
    DateTimePicker (215,185 230x30)
        p2234502574: FB_PublicHoliday.astPublicHoliday[28].datDate
        p1880513200: dd.MM.yyyy
    Rectangle (215,230 230x30)
    DateTimePicker (215,230 230x30)
        p2234502574: FB_PublicHoliday.astPublicHoliday[29].datDate
        p1880513200: dd.MM.yyyy
END_VISUALIZATION

// Device/Application/Visu/2_Clock Settings/Clock_Holiday
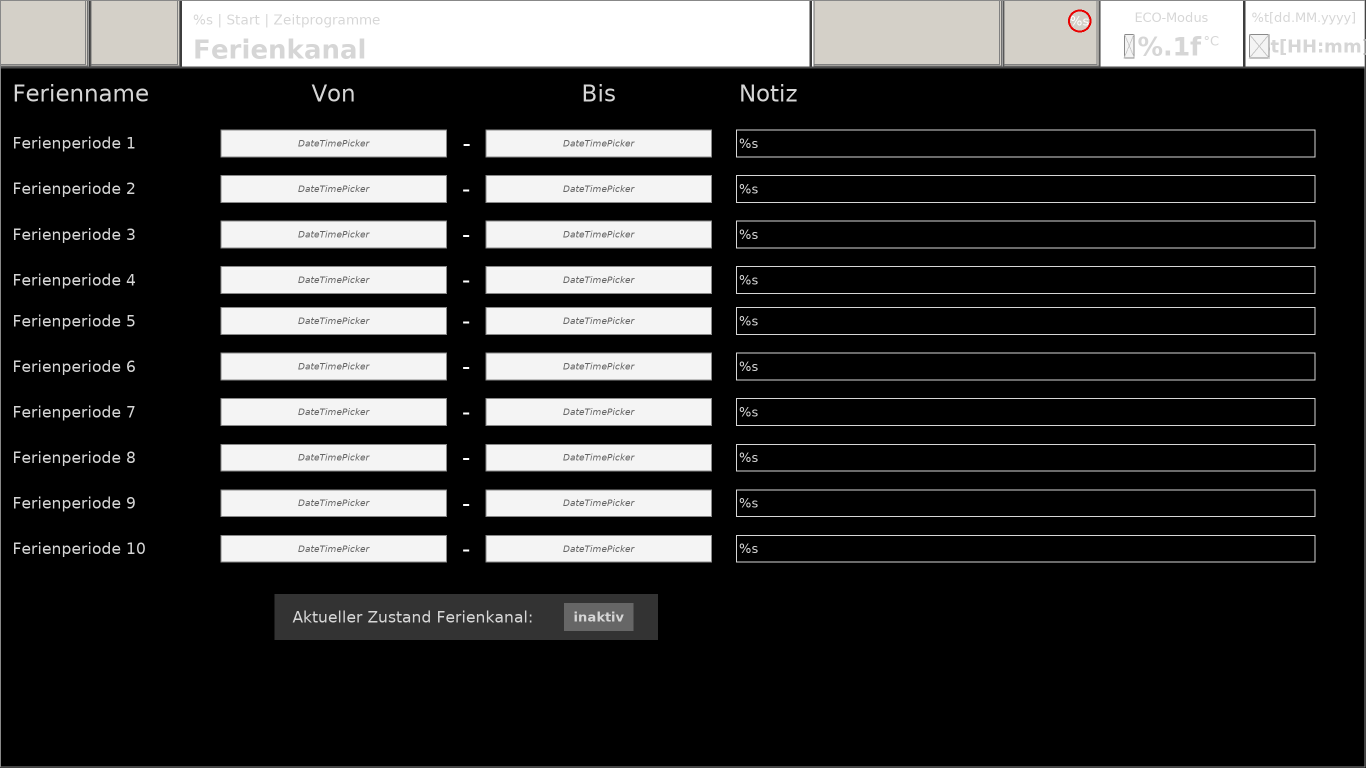
VISUALIZATION Clock_Holiday  // 1366x768
    Frame (0,0 1366x70)
        shows Header_Frame()
    Rectangle (190,5 545x30), "%s | Start | Zeitprogramme", text variable: PRG.GebVar
    Rectangle (190,32 545x35), "Ferienkanal"
    Rectangle (150,150 300x250)
    Rectangle (150,175 300x30), "PERSISTENCE"
    Image (235,230 126x125), image: HVACV.HVACImage.book
    Button (150,150 300x250)
        OnMouseClick:  Assign=Settings_Persistence, Type=Assignment
    Rectangle (530,150 300x250)
    Rectangle (530,175 300x30), "MAN INFO"
    Image (635,230 96x96), image: HVACV.HVACImage.edit2
    RoundedRectangle (620,350 120x30), "inaktiv", invisible if: Main.ManInfo.xManActive
    RoundedRectangle (620,350 120x30), "aktiv", invisible if: NOT Main.ManInfo.xManActive
    Button (530,150 300x250)
        OnMouseClick:  Assign=Settings_MANInfo, Type=Assignment
    Frame (0,75 1341x636)
        shows Holiday(FB_Holiday := PRG.Holiday_Demo)
END_VISUALIZATION

// Device/Application/Visu/2_Clock Settings/Clock_Public_Holiday
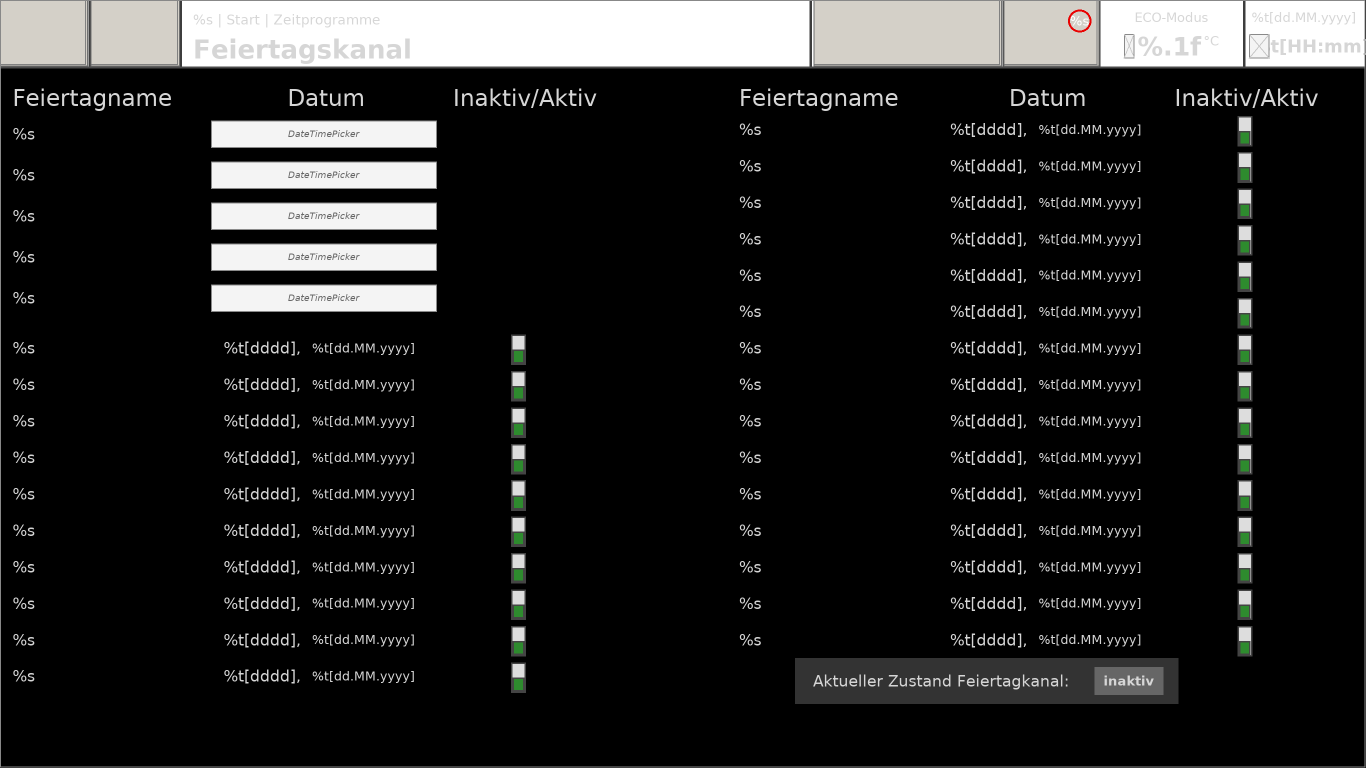
VISUALIZATION Clock_Public_Holiday  // 1366x768
    Frame (0,0 1366x70)
        shows Header_Frame()
    Rectangle (190,5 545x30), "%s | Start | Zeitprogramme", text variable: PRG.GebVar
    Rectangle (190,32 545x35), "Feiertagskanal"
    Rectangle (150,150 300x250)
    Rectangle (150,175 300x30), "PERSISTENCE"
    Image (235,230 126x125), image: HVACV.HVACImage.book
    Button (150,150 300x250)
        OnMouseClick:  Assign=Settings_Persistence, Type=Assignment
    Rectangle (530,150 300x250)
    Rectangle (530,175 300x30), "MAN INFO"
    Image (635,230 96x96), image: HVACV.HVACImage.edit2
    RoundedRectangle (620,350 120x30), "inaktiv", invisible if: Main.ManInfo.xManActive
    RoundedRectangle (620,350 120x30), "aktiv", invisible if: NOT Main.ManInfo.xManActive
    Button (530,150 300x250)
        OnMouseClick:  Assign=Settings_MANInfo, Type=Assignment
    Frame (0,75 1341x636)
        shows PublicHoliday(FB_PublicHoliday := PRG.PublicHoliday_Demo)
END_VISUALIZATION

// Device/Application/Visu/2_Clock Settings/Clock_SwitchTimeS
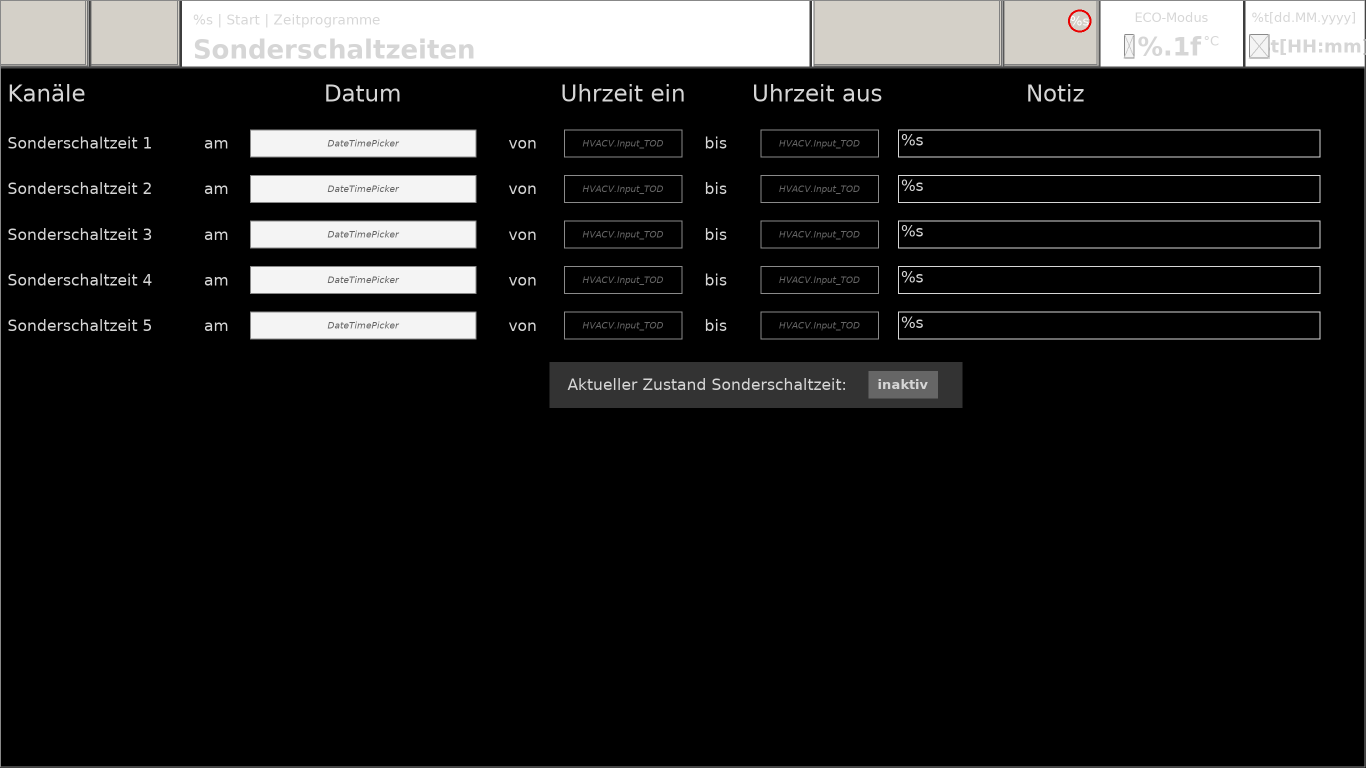
VISUALIZATION Clock_SwitchTimeS  // 1366x768
    Frame (0,0 1366x70)
        shows Header_Frame()
    Rectangle (190,5 545x30), "%s | Start | Zeitprogramme", text variable: PRG.GebVar
    Rectangle (190,32 545x35), "Sonderschaltzeiten"
    Rectangle (150,150 300x250)
    Rectangle (150,175 300x30), "PERSISTENCE"
    Image (235,230 126x125), image: HVACV.HVACImage.book
    Button (150,150 300x250)
        OnMouseClick:  Assign=Settings_Persistence, Type=Assignment
    Rectangle (530,150 300x250)
    Rectangle (530,175 300x30), "MAN INFO"
    Image (635,230 96x96), image: HVACV.HVACImage.edit2
    RoundedRectangle (620,350 120x30), "inaktiv", invisible if: Main.ManInfo.xManActive
    RoundedRectangle (620,350 120x30), "aktiv", invisible if: NOT Main.ManInfo.xManActive
    Button (530,150 300x250)
        OnMouseClick:  Assign=Settings_MANInfo, Type=Assignment
    Frame (0,75 1341x636)
        shows SwitchTimeS(FB_SwitchTimeS := PRG.SwitchTimeS_Demo)
END_VISUALIZATION

// Device/Application/Macros and frames/Clock/SwitchTimeS
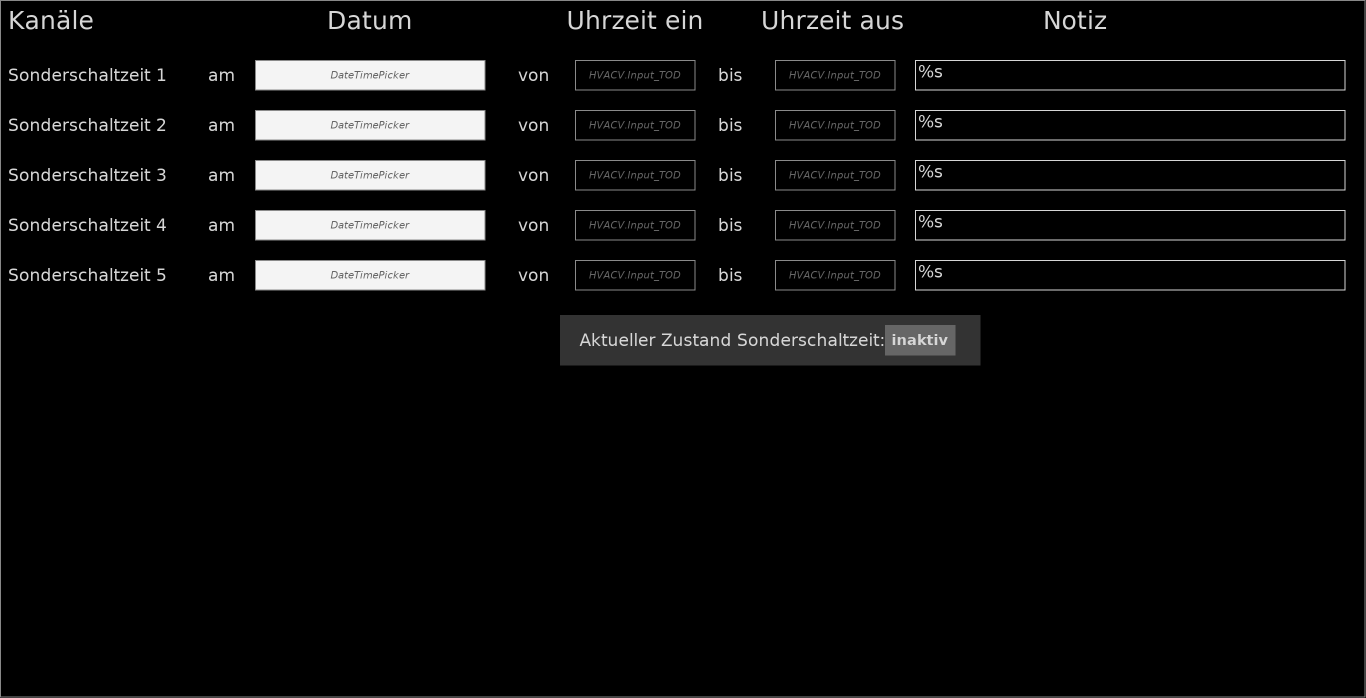
VISUALIZATION SwitchTimeS  // 1366x698
VAR_IN_OUT
	FB_SwitchTimeS : HVAC.SwitchTimeS;
END_VAR
    Rectangle (5,60 200x30), "Sonderschaltzeit 1"
    Rectangle (515,60 55x30), "von"
    Rectangle (715,60 55x30), "bis"
    Rectangle (205,60 45x30), "am"
    Rectangle (5,5 235x30), "Kanäle"
    Rectangle (255,5 230x30), "Datum"
    Rectangle (755,5 155x30), "Uhrzeit aus"
    Rectangle (560,5 150x30), "Uhrzeit ein"
    Rectangle (5,110 200x30), "Sonderschaltzeit 2"
    Rectangle (515,110 55x30), "von"
    Rectangle (715,110 55x30), "bis"
    Rectangle (205,110 45x30), "am"
    Rectangle (915,60 430x30), "%s", text variable: FB_SwitchTimeS.sCH1_Notice
        OnMouseClick: write the text variable via Default
    Rectangle (915,110 430x30), "%s", text variable: FB_SwitchTimeS.sCH2_Notice
        OnMouseClick: write the text variable via Default
    Rectangle (915,5 320x30), "Notiz"
    Rectangle (5,160 200x30), "Sonderschaltzeit 3"
    Rectangle (515,160 55x30), "von"
    Rectangle (715,160 55x30), "bis"
    Rectangle (205,160 45x30), "am"
    Rectangle (5,210 200x30), "Sonderschaltzeit 4"
    Rectangle (515,210 55x30), "von"
    Rectangle (715,210 55x30), "bis"
    Rectangle (205,210 45x30), "am"
    Rectangle (915,160 430x30), "%s", text variable: FB_SwitchTimeS.sCH3_Notice
        OnMouseClick: write the text variable via Default
    Rectangle (915,210 430x30), "%s", text variable: FB_SwitchTimeS.sCH4_Notice
        OnMouseClick: write the text variable via Default
    Rectangle (5,260 200x30), "Sonderschaltzeit 5"
    Rectangle (515,260 55x30), "von"
    Rectangle (715,260 55x30), "bis"
    Rectangle (205,260 45x30), "am"
    Rectangle (915,260 430x30), "%s", text variable: FB_SwitchTimeS.sCH5_Notice
        OnMouseClick: write the text variable via Default
    Rectangle (560,315 420x50), "Aktueller Zustand Sonderschaltzeit:"
    RoundedRectangle (895,325 50x30), "aktiv", invisible if: NOT(FB_SwitchTimeS.xActive)
    RoundedRectangle (885,325 70x30), "inaktiv", invisible if: FB_SwitchTimeS.xActive
    Frame (575,60 120x30)
        shows HVACV.Input_TOD(todTimeOfDay := FB_SwitchTimeS.todCH1_TimeFrom)
    Frame (775,60 120x30)
        shows HVACV.Input_TOD(todTimeOfDay := FB_SwitchTimeS.todCH1_TimeTo)
    Rectangle (255,60 230x30)
    DateTimePicker (255,60 230x30)
        p2234502574: FB_SwitchTimeS.datCH1_Date
        p1880513200: dd.MM.yyyy
    Rectangle (255,110 230x30)
    DateTimePicker (255,110 230x30)
        p2234502574: FB_SwitchTimeS.datCH2_Date
        p1880513200: dd.MM.yyyy
    Rectangle (255,160 230x30)
    DateTimePicker (255,160 230x30)
        p2234502574: FB_SwitchTimeS.datCH3_Date
        p1880513200: dd.MM.yyyy
    Rectangle (255,210 230x30)
    DateTimePicker (255,210 230x30)
        p2234502574: FB_SwitchTimeS.datCH4_Date
        p1880513200: dd.MM.yyyy
    Rectangle (255,260 230x30)
    DateTimePicker (255,260 230x30)
        p2234502574: FB_SwitchTimeS.datCH5_Date
        p1880513200: dd.MM.yyyy
    Frame (775,110 120x30)
        shows HVACV.Input_TOD(todTimeOfDay := FB_SwitchTimeS.todCH2_TimeTo)
    Frame (575,110 120x30)
        shows HVACV.Input_TOD(todTimeOfDay := FB_SwitchTimeS.todCH2_TimeFrom)
    Frame (775,160 120x30)
        shows HVACV.Input_TOD(todTimeOfDay := FB_SwitchTimeS.todCH3_TimeTo)
    Frame (575,160 120x30)
        shows HVACV.Input_TOD(todTimeOfDay := FB_SwitchTimeS.todCH3_TimeFrom)
    Frame (775,210 120x30)
        shows HVACV.Input_TOD(todTimeOfDay := FB_SwitchTimeS.todCH4_TimeTo)
    Frame (575,210 120x30)
        shows HVACV.Input_TOD(todTimeOfDay := FB_SwitchTimeS.todCH4_TimeFrom)
    Frame (775,260 120x30)
        shows HVACV.Input_TOD(todTimeOfDay := FB_SwitchTimeS.todCH5_TimeTo)
    Frame (575,260 120x30)
        shows HVACV.Input_TOD(todTimeOfDay := FB_SwitchTimeS.todCH5_TimeFrom)
END_VISUALIZATION

// Device/Application/Visu/1_Objects/Objects_Start
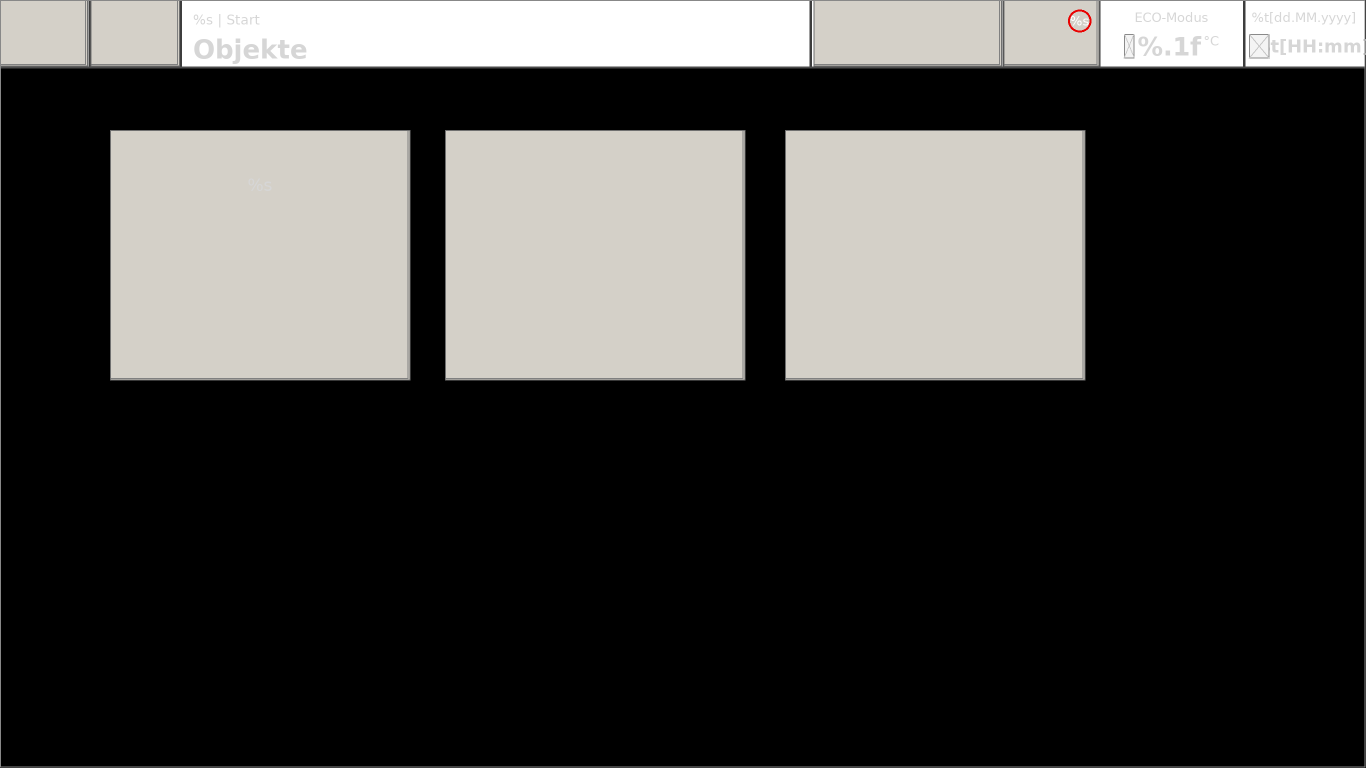
VISUALIZATION Objects_Start  // 1366x768
    Rectangle (110,130 300x250)
    Rectangle (110,140 300x30), "%s", text variable: PRG.HC_1.Title
    Image (205,205 112x112), image: HVACV.HVACImage.heating_circuit
    RoundedRectangle (220,335 79x30), "Störung", invisible if: NOT(PRG.HC_1.STATUS_ALARM)
    RoundedRectangle (225,335 71x30), "hand", invisible if: PRG.HC_1.STATUS_AUTO OR PRG.HC_1.STATUS_ALARM
    RoundedRectangle (205,335 114x30), "Automatik", invisible if: (NOT PRG.HC_1.STATUS_AUTO) OR PRG.HC_1.STATUS_ALARM
    Button (110,130 300x250)
        OnMouseClick:  Assign=Start_HC_1, Type=Assignment
    Rectangle (110,170 300x30), "%s", text variable: PRG.HC_1.Line1
    Frame (0,0 1366x70)
        shows Header_Frame()
    Rectangle (190,5 545x30), "%s | Start", text variable: PRG.GebVar
    Rectangle (190,32 545x35), "Objekte"
    Rectangle (445,130 300x250)
    Rectangle (445,140 300x30), "%s", text variable: PRG.Room_1.Titel
    Image (545,215 101x86), image: HVACV.HVACImage.room
    RoundedRectangle (555,335 79x30), "Störung", invisible if: NOT(PRG.Room_1.STATUS_SSM)
    Rectangle (445,170 300x30), "%s", text variable: PRG.Room_1.Zeile1
    RoundedRectangle (560,335 71x30), "hand", invisible if: PRG.Room_1.STATUS_AUTO OR PRG.Room_1.STATUS_SSM
    RoundedRectangle (540,335 114x30), "Automatik", invisible if: (NOT PRG.Room_1.STATUS_AUTO) OR PRG.Room_1.STATUS_SSM
    Button (445,130 300x250)
        OnMouseClick:  Assign=Start_Room_1, Type=Assignment
    Rectangle (785,130 300x250)
    Rectangle (785,140 300x30), "%s", text variable: PRG.AHU_1.Title
    Image (885,215 96x95), image: HVACV.HVACImage.fan2
    Rectangle (785,170 300x30), "%s", text variable: PRG.AHU_1.Line1
    RoundedRectangle (895,330 79x30), "Störung", invisible if: NOT(PRG.AHU_1.STATUS_ALARM)
    RoundedRectangle (900,330 71x30), "hand", invisible if: PRG.AHU_1.STATUS_AUTO OR PRG.AHU_1.STATUS_ALARM
    RoundedRectangle (880,330 114x30), "Automatik", invisible if: (NOT PRG.AHU_1.STATUS_AUTO) OR PRG.AHU_1.STATUS_ALARM
    Button (785,130 300x250)
        OnMouseClick:  Assign=Start_AHU_1, Type=Assignment
END_VISUALIZATION

// Device/Application/Visu/4_Weather/Weather_Start
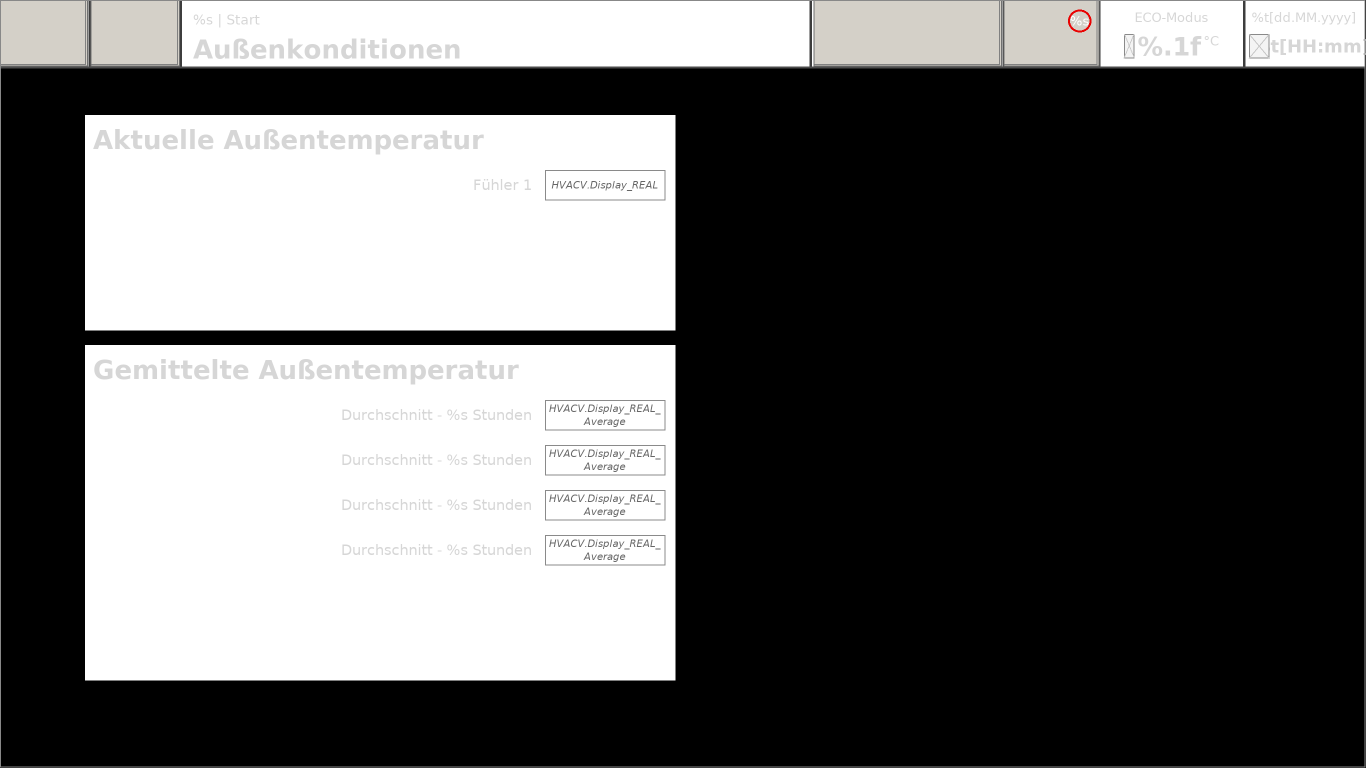
VISUALIZATION Weather_Start  // 1366x768
    Frame (0,0 1366x70)
        shows Header_Frame()
    Rectangle (190,5 545x30), "%s | Start", text variable: PRG.GebVar
    Rectangle (190,32 545x35), "Außenkonditionen"
    Rectangle (85,345 590x335)
    Rectangle (90,350 570x40), "Gemittelte Außentemperatur"
    Rectangle (85,400 450x30), "Durchschnitt - %s Stunden", text variable: Main.AverageTime.wCH0Time
    Rectangle (85,115 590x215)
    Rectangle (90,120 570x40), "Aktuelle Außentemperatur"
    Rectangle (85,170 450x30), "Fühler 1"
    Frame (545,170 120x30)
        shows HVACV.Display_REAL(rValue := Main.OutsideTemp_TS, bDecimals := 1, xAlarm := Main.OutsideTemp_TS_ERR, sUnit := '°C')
    Frame (545,400 120x30)
        shows HVACV.Display_REAL_Average(rValue := Main.AverageTime.rOutCH0, bDecimals := 1, sUnit := '°C')
    Rectangle (85,445 450x30), "Durchschnitt - %s Stunden", text variable: Main.AverageTime.wCH1Time
    Frame (545,445 120x30)
        shows HVACV.Display_REAL_Average(rValue := Main.AverageTime.rOutCH1, bDecimals := 1, sUnit := '°C')
    Rectangle (85,490 450x30), "Durchschnitt - %s Stunden", text variable: Main.AverageTime.wCH2Time
    Frame (545,490 120x30)
        shows HVACV.Display_REAL_Average(rValue := Main.AverageTime.rOutCH2, bDecimals := 1, sUnit := '°C')
    Rectangle (85,535 450x30), "Durchschnitt - %s Stunden", text variable: Main.AverageTime.wCH3Time
    Frame (545,535 120x30)
        shows HVACV.Display_REAL_Average(rValue := Main.AverageTime.rOutCH3, bDecimals := 1, sUnit := '°C')
END_VISUALIZATION

// Device/Application/Visu/1_Objects/AHU_1/Start_AHU_1
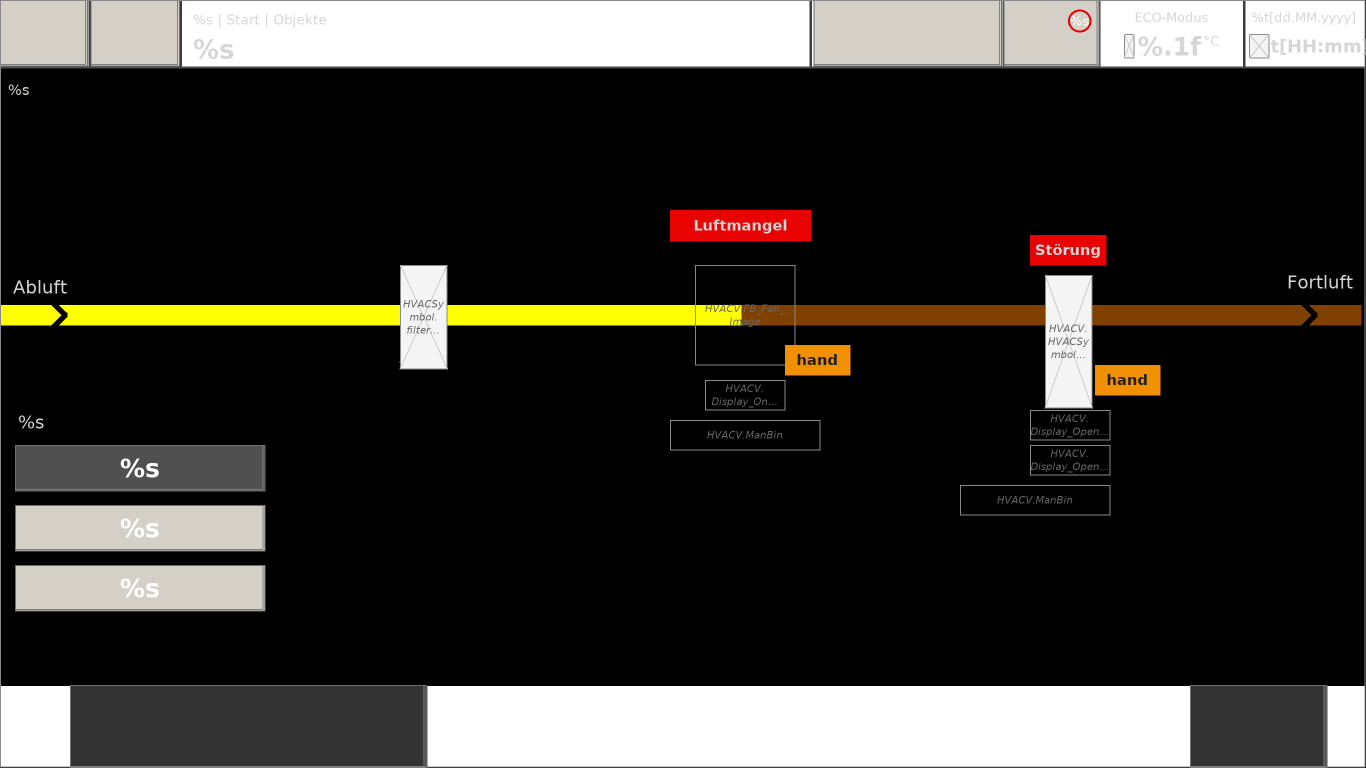
VISUALIZATION Start_AHU_1  // 1366x768
    Frame (0,0 1366x70)
        shows Header_Frame()
    Rectangle (190,5 545x30), "%s | Start | Objekte", text variable: PRG.GebVar
    Rectangle (190,32 545x35), "%s", text variable: PRG.AHU_1.Title
    Rectangle (0,685 1366x83)
    Rectangle (425,685 2x83)
    Rectangle (70,685 2x83)
    Rectangle (130,685 166x83), "ZEITSCHALTUNG"
    Image (80,710 36x35), image: HVACV.HVACImage.clock
    RoundedRectangle (295,710 120x30), "inaktiv", invisible if: PRG.AHU_1.Clock.xActive
    RoundedRectangle (295,710 120x30), "aktiv", invisible if: NOT PRG.AHU_1.Clock.xActive
    Button (70,685 356x83)
        OnMouseClick:  Assign=Clock_AHU_1, Type=Assignment
    Rectangle (1190,685 2x83)
    Rectangle (1325,685 2x83)
    Rectangle (1260,685 71x83), "HILFE"
    Image (1205,705 31x47), image: HVACV.HVACImage.help
    Button (1190,685 136x83)
        OnMouseClick:  Dialog=HVACV.Help_Start, OpenModal=True, OpenCentered=True
    Frame (0,70 1366x613)
        shows ExhaustAir(FB := PRG.AHU_1)
END_VISUALIZATION

// Device/Application/Macros and frames/Exhaust air system/ExhaustAir
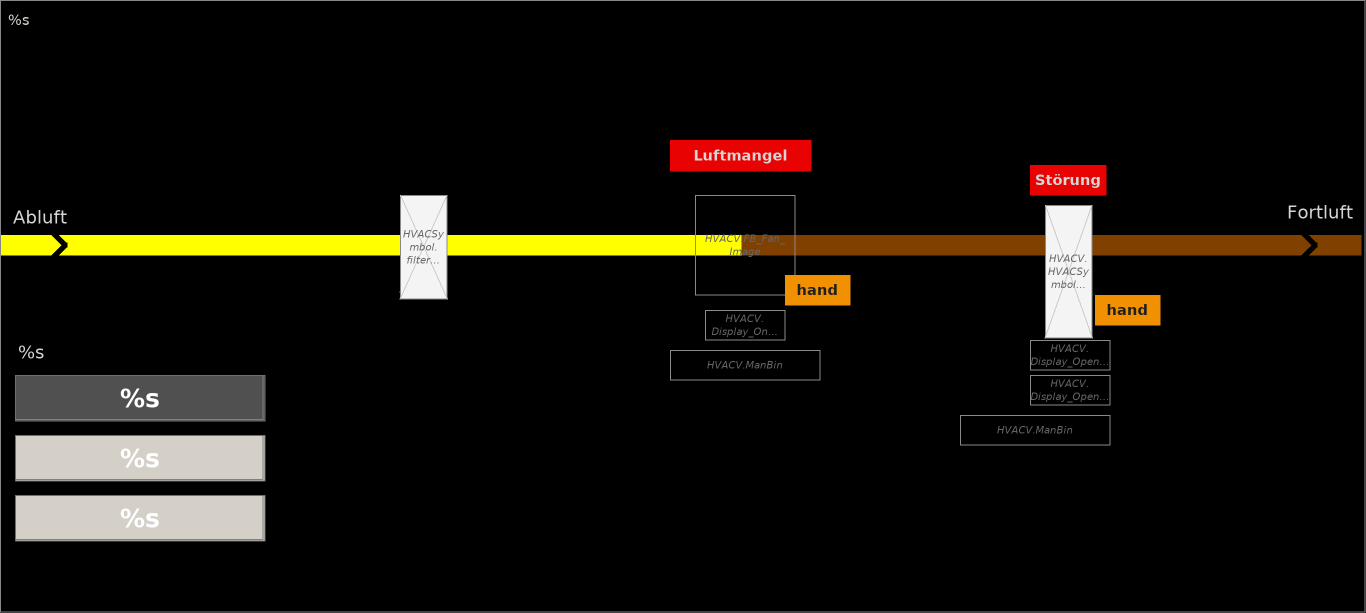
VISUALIZATION ExhaustAir  // 1366x613
VAR_IN_OUT
	FB : ExhaustAir ;
END_VAR
    Rectangle (730,235 631x20)
    Rectangle (5,0 970x40), "%s", text variable: FB.Line1
    Rectangle (0,235 741x20)
    Polyline (50,230) (65,245) (50,260)
    Polyline (1300,230) (1315,245) (1300,260)
    Button (15,375 250x46), "%s", text variable: FB.OS.sTitleM0, colour toggle: FB.OS.eMode = 0
        OnMouseClick: execute { FB.OS.eMode := 0; }
    Button (15,435 250x46), "%s", text variable: FB.OS.sTitleM1, colour toggle: FB.OS.eMode =1
        OnMouseClick: execute { FB.OS.eMode := 1; }
    Button (15,495 250x46), "%s", text variable: FB.OS.sTitleM2, colour toggle: FB.OS.eMode =2
        OnMouseClick: execute { FB.OS.eMode := 2; }
    Rectangle (15,340 251x25), "%s", text variable: FB.OS.sTitle
    Rectangle (1210,200 146x25), "Fortluft"
    Image (1045,205 47x133), image: HVACV.HVACSymbol.damper_vertical_Mbottom
    Rectangle (10,205 171x25), "Abluft"
    Frame (695,195 100x100)
        shows HVACV.FB_Fan_Image(xFeedback := FB.Fan_Fb, xAlarm := FB.Fan.xAlarm, iRotation := 90)
    Frame (1030,375 80x30)
        shows HVACV.Display_Open_Close(OpenFeedback := FB.OA_OPEN, CloseFeedback := FB.OA_CLOSE)
    Frame (1030,340 80x30)
        shows HVACV.Display_Open_Close_Setpoint(Setpoint := FB.Damper_HB)
    Frame (960,415 150x30)
        shows HVACV.ManBin(eManModeB := FB.Damper_OutsideAir.eManModeB)
    Frame (705,310 80x30)
        shows HVACV.Display_On_Off_Setpoint(Setpoint := FB.Fan_HB)
    Frame (670,350 150x30)
        shows HVACV.ManBin(eManModeB := FB.Fan.eManModeB)
    RoundedRectangle (670,140 141x31), "Luftmangel", invisible if: FB.Fan.xPFb
    RoundedRectangle (785,275 65x30), "hand", invisible if: FB.Fan_AOO = 0
    RoundedRectangle (1095,295 65x30), "hand", invisible if: FB.OA_Damper_AOO = 0
    Image (400,195 45x97), image: HVACSymbol.filter
    Image (400,195 47x104), invisible if: NOT FB.FilterMonitoringB.xAlarm, image: HVACSymbol.filter_caution
    RoundedRectangle (1030,165 76x30), "Störung", invisible if: NOT FB.Damper_OutsideAir.xAlarm
END_VISUALIZATION

// Device/Application/Visu/1_Objects/AHU_1/Clock_AHU_1
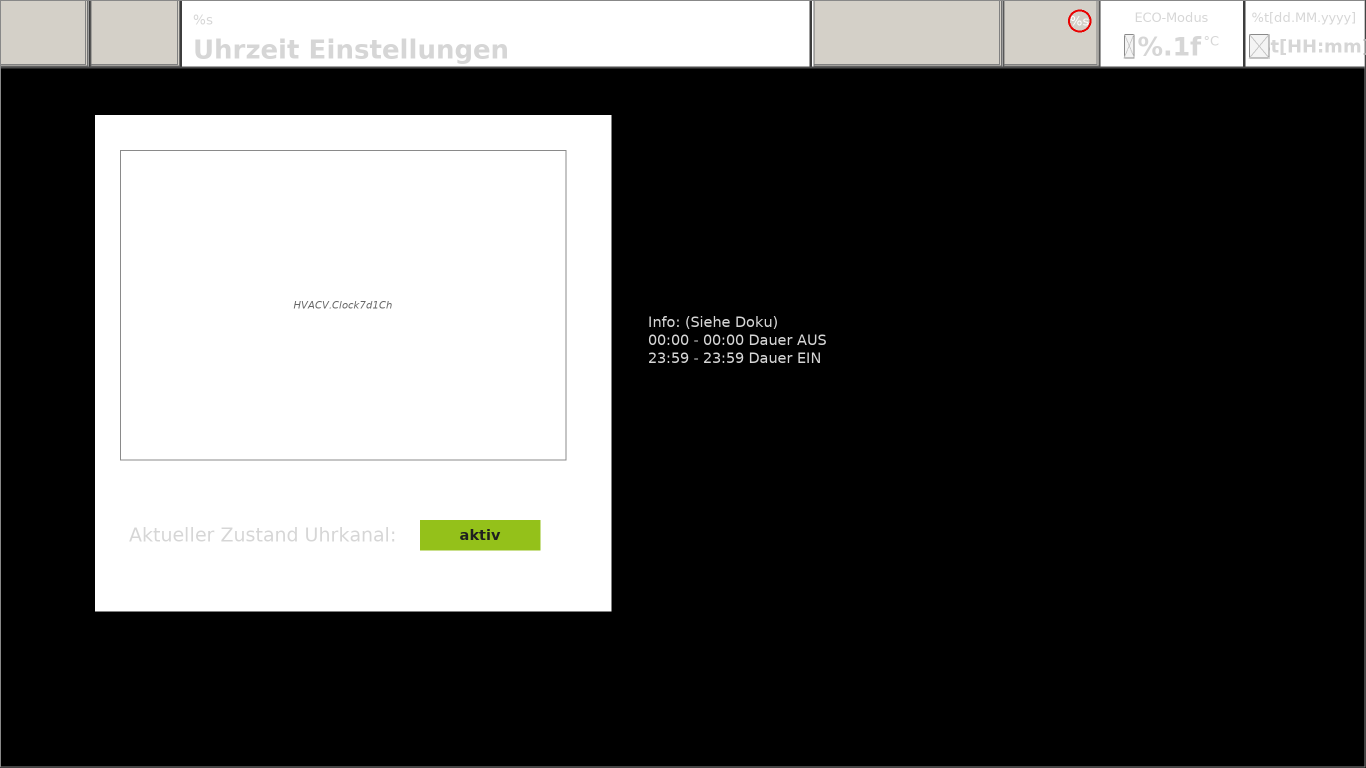
VISUALIZATION Clock_AHU_1  // 1366x768
    Rectangle (95,115 516x496)
    Frame (0,0 1366x70)
        shows Header_Frame()
    Rectangle (190,5 545x30), "%s", text variable: CONCAT( CONCAT(PRG.GebVar, ' | Start | Objekte | '), Prg.AHU_1.Title)
    Rectangle (190,32 545x35), "Uhrzeit Einstellungen", text variable: PRG.AHU_1.Title
    RoundedRectangle (420,520 120x30), "inaktiv", invisible if: PRG.AHU_1.Clock.xActive
    RoundedRectangle (420,520 120x30), "aktiv", invisible if: NOT PRG.AHU_1.Clock.xActive
    Rectangle (115,520 296x30), "Aktueller Zustand Uhrkanal:"
    Frame (120,150 446x310)
        shows HVACV.Clock7d1Ch(FB_Clock7d1Ch := PRG.AHU_1.Clock)
    Rectangle (645,295 447x90), "Info: (Siehe Doku) 00:00 - 00:00 Dauer AUS 23:59 - 23:59 Dauer EIN"
END_VISUALIZATION

(* text list AlarmGroup (id | default | EN)
  25 | RLT1: Außenluftklappe auf Handbetrieb (Hardware) | AHU1: Exhaust air damper on manual mode (Hardware)
  24 | RLT1: Ventilator auf Handbetrieb (Hardware) | AHU1: Fan on manual mode (Hardware)
  23 | RLT1: Ventilator auf Handbetrieb (Software) | AHU1: Fan on manual mode (Software)
  22 | RLT1: Außenluftklappe auf Handbetrieb (Software) | AHU1: Exhaust air damper on manual mode (Software)
  21 | RLT1: Anlagenschalter auf Handbetrieb | AHU1: Operation mode selector on manual mode
  20 | RLT1: Abluftfilter Wartung notwendig | AHU1: Exhaust filter service
  19 | RLT1: Abluftventilator | AHU1: Exhaust Fan
  18 | RLT1: Außenluftklappe Störung | RLT: Exhaust air damper error
  17 | Room 1: Ventil auf Handbetrieb (Software) | Room1: Valve on manual mode (Software)
  16 | Room 1: Ventil auf Handbetrieb (Hardware) | Room1: Valve on manual mode (Hardware)
  15 | Room 1: Anlagenschalter Betriebsmodus auf Handbetrieb | Room1: Operation mode selector on manual mode
  14 | Room 1: Frostgefahr | Room1: Frost danger
  13 | Room 1: Raumtemperaturfühler Wert gestört | Room1: Room temperature sensor value error
  12 | Heizkreis 1: Anlagenwahlschalter auf Handbetrieb (Software) | Heat circuit 1: Operation mode selector on manual mode
  10 | Heizkreis 1: Pumpe auf Handbetrieb (Software) | Heat circuit 1:  Pump on manual mode (Software)
  11 | Heizkreis 1: Ventil auf Handbetrieb (Software) | Heat circuit 1:  Valve on manual mode (Software)
  9 | Heizkreis 1: Ventil auf Handbetrieb (Hardware) | Heat circuit 1:  Valve on manual mode (Hardware)
  8 | Heizkreis 1: Pumpe auf Handbetrieb (Hardware) | Heat circuit 1:  Pump on manual mode (Hardware)
  7 | Heizkreis 1: Ventil | Heat circuit 1: Valve
  6 | Heizkreis 1:  Rücklauftemperaturfühler Wert gestört | Heat circuit 1: Return temperature sensor value error
  5 | Heizkreis 1:  Vorlauftemperaturfühler Wert gestört | Heat circuit 1: Flow temperature sensor value error
  4 | Heizkreis 1: Pumpe Betriebsüberwachung | Heat circuit 1: Pump feedback control
  3 | Heizkreis 1: Pumpe | Heat circuit 1: Pump
  2 | Test Alarm Class Warning | 
  1 | Test Alarm Class Info | 
  0 | Test Alarm Class Error | 
   |  |  *)

(* text list System (id | default | de)
  Apr | Apr | 
  April | April | April
  Aug | Aug | Aug
  August | August | August
  Dec | Dec | Dez
  December | December | Dezember
  Feb | Feb | Feb
  February | February | Februar
  Fri | Fri | Fr
  Friday | Friday | Freitag
  Jan | Jan | Jan
  January | January | Januar
  Jul | Jul | Jul
  July | July | Juli
  Jun | Jun | Jun
  June | June | Juni
  Mar | Mar | Mär
  March | March | März
  May | May | Mai
  May_3Letter | May | Mai
  Mon | Mon | Mo
  Monday | Monday | Montag
  Nov | Nov | Nov
  November | November | November
  Oct | Oct | Okt
  October | October | Oktober
  Sat | Sat | Sa
  Saturday | Saturday | Samstag
  Sep | Sep | Sep
  September | September | September
  Sun | Sun | So
  Sunday | Sunday | Sonntag
  Thu | Thu | Do
  Thursday | Thursday | Donnerstag
  Tue | Tue | Di
  Tuesday | Tuesday | Dienstag
  Wed | Wed | Mi
  Wednesday | Wednesday | Mittwoch
   |  |  *)

(* text PersistenceConfig
// Persistence configuration for application Device.Application
// Generated automatically by GenPersistence
SEC General
  Application := Device.Application ;
  ExcludedGroups := [  ] ;
  ToplevelInstanceNames := [ PersistenceManager ] ;
  ToplevelFBPaths := [ GVL_PersistenceManager.PersistenceManager ] ;
END_SEC
SEC Channel : HVAC_Parameter
  Groups := [ HVAC_Parameter ] ;
  FBPath := PersistenceManager.INST_HVAC_Parameter ;
  SeparateArchivePerToplevelInstance := False ;
  CompressTags := True ;
  MaximumFileSize := 0 ;
END_SEC
SEC Channel : HVAC_Counter
  Groups := [ HVAC_Counter ] ;
  FBPath := PersistenceManager.INST_HVAC_Counter ;
  SeparateArchivePerToplevelInstance := False ;
  CompressTags := True ;
  MaximumFileSize := 0 ;
END_SEC
*)
